W262.13 BOOL  ; B3右伺服位置8设置（HMI）
W262.14 BOOL  ; B3右伺服位置9设置（HMI）
W262.15 BOOL  ; B3右伺服位置10设置（HMI）
W263.00 BOOL  ; B3右伺服待机位手动(HMI)
W263.01 BOOL  ; B3右伺服拨料退回位手动(HMI)
W263.02 BOOL  ; B3右伺服拨料位手动(HMI)
W263.03 BOOL  ; B3右伺服减速位手动(HMI)
W263.04 BOOL  ; B3右伺服等距热压位手动(HMI)
W263.05 BOOL  ; B3右伺服位置6手动(HMI)
W263.06 BOOL  ; B3右伺服位置7手动(HMI)
W263.07 BOOL  ; B3右伺服位置8手动(HMI)
W263.08 BOOL  ; B3右伺服位置9手动(HMI)
W263.09 BOOL  ; B3右伺服位置10手动(HMI)
W263.10 BOOL  ; B3右伺服回原条件
W263.11 BOOL  ; B3右伺服运行锁定
W263.12 BOOL  ; B3右伺服定位条件
W263.13 BOOL  ; B3右伺服回原启动
W263.14 BOOL  ; B3右伺服回原完成
W263.15 BOOL  ; B3右伺服辅助3
W264.00 BOOL  ; B4左伺服回原点手动(HMI)
W264.01 BOOL  ; B4左伺服错误清除(HMI)
W264.02 BOOL  ; B4左伺服JOG高速(HMI)
W264.03 BOOL  ; B4左伺服JOG低速（（HMI）
W264.04 BOOL  ; B4左伺服JOG+（HMI）
W264.05 BOOL  ; B4左伺服JOG-（HMI）
W264.06 BOOL  ; B4左伺服待机位设置（HMI）
W264.07 BOOL  ; B4左伺服拨料退回位设置（HMI）
W264.08 BOOL  ; B4左伺服拨料位设置（HMI）
W264.09 BOOL  ; B4左伺服减速位设置（HMI）
W264.10 BOOL  ; B4左伺服等距热压位设置（HMI）
W264.11 BOOL  ; B4左伺服位置6设置（HMI）
W264.12 BOOL  ; B4左伺服位置7设置（HMI）
W264.13 BOOL  ; B4左伺服位置8设置（HMI）
W264.14 BOOL  ; B4左伺服位置9设置（HMI）
W264.15 BOOL  ; B4左伺服位置10设置（HMI）
W265.00 BOOL  ; B4左伺服待机位手动(HMI)
W265.01 BOOL  ; B4左伺服拨料退回位手动(HMI)
W265.02 BOOL  ; B4左伺服拨料位手动(HMI)
W265.03 BOOL  ; B4左伺服减速位手动(HMI)
W265.04 BOOL  ; B4左伺服等距热压位手动(HMI)
W265.05 BOOL  ; B4左伺服位置6手动(HMI)
W265.06 BOOL  ; B4左伺服位置7手动(HMI)
W265.07 BOOL  ; B4左伺服位置8手动(HMI)
W265.08 BOOL  ; B4左伺服位置9手动(HMI)
W265.09 BOOL  ; B4左伺服位置10手动(HMI)
W265.10 BOOL  ; B4左伺服回原条件
W265.11 BOOL  ; B4左伺服运行锁定
W265.12 BOOL  ; B4左伺服定位条件
W265.13 BOOL  ; B4左伺服回原启动
W265.14 BOOL  ; B4左伺服回原完成
W265.15 BOOL  ; B4左伺服辅助3
W266.00 BOOL  ; B4右伺服回原点手动(HMI)
W266.01 BOOL  ; B4右伺服错误清除(HMI)
W266.02 BOOL  ; B4右伺服JOG高速(HMI)
W266.03 BOOL  ; B4右伺服JOG低速（（HMI）
W266.04 BOOL  ; B4右伺服JOG+（HMI）
W266.05 BOOL  ; B4右伺服JOG-（HMI）
W266.06 BOOL  ; B4右伺服待机位设置（HMI）
W266.07 BOOL  ; B4右伺服拨料退回位设置（HMI）
W266.08 BOOL  ; B4右伺服拨料位设置（HMI）
W266.09 BOOL  ; B4右伺服减速位设置（HMI）
W266.10 BOOL  ; B4右伺服等距热压位设置（HMI）
W266.11 BOOL  ; B4右伺服位置6设置（HMI）
W266.12 BOOL  ; B4右伺服位置7设置（HMI）
W266.13 BOOL  ; B4右伺服位置8设置（HMI）
W266.14 BOOL  ; B4右伺服位置9设置（HMI）
W266.15 BOOL  ; B4右伺服位置10设置（HMI）
W267.00 BOOL  ; B4右伺服待机位手动(HMI)
W267.01 BOOL  ; B4右伺服拨料退回位手动(HMI)
W267.02 BOOL  ; B4右伺服拨料位手动(HMI)
W267.03 BOOL  ; B4右伺服减速位手动(HMI)
W267.04 BOOL  ; B4右伺服等距热压位手动(HMI)
W267.05 BOOL  ; B4右伺服位置6手动(HMI)
W267.06 BOOL  ; B4右伺服位置7手动(HMI)
W267.07 BOOL  ; B4右伺服位置8手动(HMI)
W267.08 BOOL  ; B4右伺服位置9手动(HMI)
W267.09 BOOL  ; B4右伺服位置10手动(HMI)
W267.10 BOOL  ; B4右伺服回原条件
W267.11 BOOL  ; B4右伺服运行锁定
W267.12 BOOL  ; B4右伺服定位条件
W267.13 BOOL  ; B4右伺服回原启动
W267.14 BOOL  ; B4右伺服回原完成
W267.15 BOOL  ; B4右伺服辅助3
W268.00 BOOL  ; 出料伸缩伺服A回原点手动(HMI)
W268.01 BOOL  ; 出料伸缩伺服A错误清除(HMI)
W268.02 BOOL  ; 出料伸缩伺服AJOG高速(HMI)
W268.03 BOOL  ; 出料伸缩伺服AJOG低速（（HMI）
W268.04 BOOL  ; 出料伸缩伺服AJOG+（HMI）
W268.05 BOOL  ; 出料伸缩伺服AJOG-（HMI）
W268.06 BOOL  ; 出料伸缩伺服A位置1设置（HMI）
W268.07 BOOL  ; 出料伸缩伺服A位置2设置（HMI）
W268.08 BOOL  ; 出料伸缩伺服A位置3设置（HMI）
W268.09 BOOL  ; 出料伸缩伺服A位置4设置（HMI）
W268.10 BOOL  ; 出料伸缩伺服A位置5设置（HMI）
W268.11 BOOL  ; 出料伸缩伺服A位置6设置（HMI）
W268.12 BOOL  ; 出料伸缩伺服A位置7设置（HMI）
W268.13 BOOL  ; 出料伸缩伺服A位置8设置（HMI）
W268.14 BOOL  ; 出料伸缩伺服A位置9设置（HMI）
W268.15 BOOL  ; 出料伸缩伺服A位置10设置（HMI）
W269.00 BOOL  ; 出料伸缩伺服A位置1手动(HMI)
W269.01 BOOL  ; 出料伸缩伺服A位置2手动(HMI)
W269.02 BOOL  ; 出料伸缩伺服A位置3手动(HMI)
W269.03 BOOL  ; 出料伸缩伺服A位置4手动(HMI)
W269.04 BOOL  ; 出料伸缩伺服A位置5手动(HMI)
W269.05 BOOL  ; 出料伸缩伺服A位置6手动(HMI)
W269.06 BOOL  ; 出料伸缩伺服A位置7手动(HMI)
W269.07 BOOL  ; 出料伸缩伺服A位置8手动(HMI)
W269.08 BOOL  ; 出料伸缩伺服A位置9手动(HMI)
W269.09 BOOL  ; 出料伸缩伺服A位置10手动(HMI)
W269.10 BOOL  ; 出料伸缩伺服A回原条件
W269.11 BOOL  ; 出料伸缩伺服A运行锁定
W269.12 BOOL  ; 出料伸缩伺服A定位条件
W269.13 BOOL  ; 出料伸缩伺服A回原启动
W269.14 BOOL  ; 出料伸缩伺服A回原完成
W269.15 BOOL  ; 出料伸缩伺服A辅助3
W26.00 BOOL  ; 3ST_进料夹爪上层无料状态正常
W26.01 BOOL  ; 3ST_进料夹爪下层无料状态正常
W26.02 BOOL  ; 3ST_出料夹爪上层无料状态正常
W26.03 BOOL  ; 3ST_出料夹爪下层无料状态正常
W26.04 BOOL  ; 3ST_A出料夹爪A1状态OK
W26.05 BOOL  ; 3ST_A出料夹爪A2状态OK
W26.06 BOOL  ; 3ST_A出料夹爪A3状态OK
W26.07 BOOL  ; 3ST_A出料夹爪A4状态OK
W26.08 BOOL  ; 3ST_A出料夹爪A5状态OK
W26.09 BOOL  ; A1真空正常
W26.10 BOOL  ; A2真空正常
W26.11 BOOL  ; A3真空正常
W26.12 BOOL  ; A4真空正常
W26.13 BOOL  ; A5真空正常
W26.14 BOOL  ; 3ST-A出料夹爪真空正常
W270.00 BOOL  ; 26#伺服回原点手动(HMI)
W270.01 BOOL  ; 26#伺服错误清除(HMI)
W270.02 BOOL  ; 26#伺服JOG高速(HMI)
W270.03 BOOL  ; 26#伺服JOG低速（（HMI）
W270.04 BOOL  ; 26#伺服JOG+（HMI）
W270.05 BOOL  ; 26#伺服JOG-（HMI）
W270.06 BOOL  ; 26#伺服位置1设置（HMI）
W270.07 BOOL  ; 26#伺服位置2设置（HMI）
W270.08 BOOL  ; 26#伺服位置3设置（HMI）
W270.09 BOOL  ; 26#伺服位置4设置（HMI）
W270.10 BOOL  ; 26#伺服位置5设置（HMI）
W270.11 BOOL  ; 26#伺服位置6设置（HMI）
W270.12 BOOL  ; 26#伺服位置7设置（HMI）
W270.13 BOOL  ; 26#伺服位置8设置（HMI）
W270.14 BOOL  ; 26#伺服位置9设置（HMI）
W270.15 BOOL  ; 26#伺服位置10设置（HMI）
W271.00 BOOL  ; 26#伺服位置1手动(HMI)
W271.01 BOOL  ; 26#伺服位置2手动(HMI)
W271.02 BOOL  ; 26#伺服位置3手动(HMI)
W271.03 BOOL  ; 26#伺服位置4手动(HMI)
W271.04 BOOL  ; 26#伺服位置5手动(HMI)
W271.05 BOOL  ; 26#伺服位置6手动(HMI)
W271.06 BOOL  ; 26#伺服位置7手动(HMI)
W271.07 BOOL  ; 26#伺服位置8手动(HMI)
W271.08 BOOL  ; 26#伺服位置9手动(HMI)
W271.09 BOOL  ; 26#伺服位置10手动(HMI)
W271.10 BOOL  ; 26#伺服回原条件
W271.11 BOOL  ; 26#伺服运行锁定
W271.12 BOOL  ; 26#伺服定位条件
W271.13 BOOL  ; 26#伺服回原启动
W271.14 BOOL  ; 26#伺服回原完成
W271.15 BOOL  ; 26#伺服辅助3
W272.00 BOOL  ; 27#左伺服回原点手动(HMI)
W272.01 BOOL  ; 27#左伺服错误清除(HMI)
W272.02 BOOL  ; 27#左伺服JOG高速(HMI)
W272.03 BOOL  ; 27#左伺服JOG低速（（HMI）
W272.04 BOOL  ; 27#左伺服JOG+（HMI）
W272.05 BOOL  ; 27#左伺服JOG-（HMI）
W272.06 BOOL  ; 27#左伺服位置1设置（HMI）
W272.07 BOOL  ; 27#左伺服位置2设置（HMI）
W272.08 BOOL  ; 27#左伺服位置3设置（HMI）
W272.09 BOOL  ; 27#左伺服位置4设置（HMI）
W272.10 BOOL  ; 27#左伺服位置5设置（HMI）
W272.11 BOOL  ; 27#左伺服位置6设置（HMI）
W272.12 BOOL  ; 27#左伺服位置7设置（HMI）
W272.13 BOOL  ; 27#左伺服位置8设置（HMI）
W272.14 BOOL  ; 27#左伺服位置9设置（HMI）
W272.15 BOOL  ; 27#左伺服位置10设置（HMI）
W273.00 BOOL  ; 27#左伺服位置1手动(HMI)
W273.01 BOOL  ; 27#左伺服位置2手动(HMI)
W273.02 BOOL  ; 27#左伺服位置3手动(HMI)
W273.03 BOOL  ; 27#左伺服位置4手动(HMI)
W273.04 BOOL  ; 27#左伺服位置5手动(HMI)
W273.05 BOOL  ; 27#左伺服位置6手动(HMI)
W273.06 BOOL  ; 27#左伺服位置7手动(HMI)
W273.07 BOOL  ; 27#左伺服位置8手动(HMI)
W273.08 BOOL  ; 27#左伺服位置9手动(HMI)
W273.09 BOOL  ; 27#左伺服位置10手动(HMI)
W273.10 BOOL  ; 27#左伺服回原条件
W273.11 BOOL  ; 27#左伺服运行锁定
W273.12 BOOL  ; 27#左伺服定位条件
W273.13 BOOL  ; 27#左伺服回原启动
W273.14 BOOL  ; 27#左伺服回原完成
W273.15 BOOL  ; 27#左伺服辅助3
W274.00 BOOL  ; 接料伺服回原点手动(HMI)
W274.01 BOOL  ; 接料伺服错误清除(HMI)
W274.02 BOOL  ; 接料伺服JOG高速(HMI)
W274.03 BOOL  ; 接料伺服JOG低速（（HMI）
W274.04 BOOL  ; 接料伺服JOG+（HMI）
W274.05 BOOL  ; 接料伺服JOG-（HMI）
W274.06 BOOL  ; 接料伺服出料位设置（HMI）
W274.07 BOOL  ; 接料伺服接料位设置（HMI）
W274.08 BOOL  ; 接料伺服位置3设置（HMI）
W274.09 BOOL  ; 接料伺服位置4设置（HMI）
W274.10 BOOL  ; 接料伺服位置5设置（HMI）
W274.11 BOOL  ; 接料伺服位置6设置（HMI）
W274.12 BOOL  ; 接料伺服位置7设置（HMI）
W274.13 BOOL  ; 接料伺服位置8设置（HMI）
W274.14 BOOL  ; 接料伺服位置9设置（HMI）
W274.15 BOOL  ; 接料伺服位置10设置（HMI）
W275.00 BOOL  ; 接料伺服出料位手动(HMI)
W275.01 BOOL  ; 接料伺服接料位手动(HMI)
W275.02 BOOL  ; 接料伺服位置3手动(HMI)
W275.03 BOOL  ; 接料伺服位置4手动(HMI)
W275.04 BOOL  ; 接料伺服位置5手动(HMI)
W275.05 BOOL  ; 接料伺服位置6手动(HMI)
W275.06 BOOL  ; 接料伺服位置7手动(HMI)
W275.07 BOOL  ; 接料伺服位置8手动(HMI)
W275.08 BOOL  ; 接料伺服位置9手动(HMI)
W275.09 BOOL  ; 接料伺服位置10手动(HMI)
W275.10 BOOL  ; 接料伺服回原条件
W275.11 BOOL  ; 接料伺服运行锁定
W275.12 BOOL  ; 接料伺服定位条件
W275.13 BOOL  ; 接料伺服回原启动
W275.14 BOOL  ; 接料伺服回原完成
W275.15 BOOL  ; 接料伺服辅助3
W27.00 BOOL  ; 3ST_进料夹爪上层有料状态正常
W27.01 BOOL  ; 3ST_进料夹爪下层有料状态正常
W27.02 BOOL  ; 3ST_出料夹爪上层有料状态正常
W27.03 BOOL  ; 3ST_出料夹爪下层有料状态正常
W28.12 BOOL  ; B进料平台允许取料信号
W28.13 BOOL  ; B出料平台允许放料信号
W28.14 BOOL  ; A进料平台允许取料信号
W28.15 BOOL  ; A出料平台允许放料信号
W29.00 BOOL  ; A移栽在上料安全位
W29.01 BOOL  ; 3ST_A移栽在下料安全位
W29.02 BOOL  ; 热压1A有上料需求
W29.03 BOOL  ; 热压2A有上料需求
W29.04 BOOL  ; 热压1A有下料需求
W29.05 BOOL  ; 热压2A有下料需求
W29.06 BOOL  ; 热压1A允许上料
W29.07 BOOL  ; 热压2A允许上料
W29.08 BOOL  ; 热压1A允许下料
W29.09 BOOL  ; 热压2A允许下料
W30.00 BOOL  ; 3ST_B手动切换允许输出标志
W30.01 BOOL  ; 3ST_B自动切换允许输出标志
W30.06 BOOL  ; A边无进料计时
W30.07 BOOL  ; 3ST_A B侧取料
W30.08 BOOL  ; 3ST_B B侧取料
W31.00 BOOL  ; 3ST_B进料夹爪有料标志
W31.01 BOOL  ; 3ST_B进料夹爪无料标志
W31.02 BOOL  ; 3ST_B出料夹爪有料标志
W31.03 BOOL  ; 3ST_B出料夹爪无料标志
W31.09 BOOL  ; B1真空正常
W31.10 BOOL  ; B2真空正常
W31.11 BOOL  ; B3真空正常
W31.12 BOOL  ; B4真空正常
W31.13 BOOL  ; B5真空正常
W31.14 BOOL  ; 3ST-B出料夹爪真空正常
W34.00 BOOL  ; 3ST_B移栽在上料安全位
W34.01 BOOL  ; 3ST_B移栽在下料安全位
W34.02 BOOL  ; 热压1B有上料需求
W34.03 BOOL  ; 热压2B有上料需求
W34.04 BOOL  ; 热压1B有下料需求
W35.00 BOOL  ; 4ST_A手动输出允许
W35.01 BOOL  ; 4ST_A自动输出允许
W35.03 BOOL  ; 4ST_A A侧放料准备(总)
W35.04 BOOL  ; 4ST_A A侧放料允许(总)
W35.05 BOOL  ; 4ST_A A侧取料准备(总)
W35.06 BOOL  ; 4ST_A A侧取料允许(总)
W35.07 BOOL  ; 4ST_A B侧放料准备(总)
W35.08 BOOL  ; 4ST_A B侧放料允许(总)
W35.09 BOOL  ; 4ST_A B侧取料准备(总)
W35.10 BOOL  ; 4ST_A B侧取料允许(总)
W36.00 BOOL  ; 4ST_A所有顶升缩回位
W36.01 BOOL  ; 4ST_A所有顶升伸出位
W36.02 BOOL  ; 4ST_A所有预压退回位
W36.03 BOOL  ; 4ST_A所有预压伸出位
W36.04 BOOL  ; 4ST_A HIP气缸全上位
W36.05 BOOL  ; 4ST_A HIP气缸全下位
W36.06 BOOL  ; 4ST_A气缸全原位
W36.07 BOOL  ; 4ST_A 下压板全A位
W36.08 BOOL  ; 4ST_A 下压板全B位
W36.09 BOOL  ; 4ST_A 侧压伺服均在初始位
W36.10 BOOL  ; 4ST_A 侧压均在拨料退回位
W36.11 BOOL  ; 4ST_A 侧压均在拨料位
W36.12 BOOL  ; 4ST_A 侧压启动&HIP&预压气缸后退条件
W36.13 BOOL  ; 4ST_A 侧压力全部到达区间
W36.14 BOOL  ; 4ST_A HIP全部测试完成
W36.15 BOOL  ; 4ST_A均在拨料等待位
W37.00 BOOL  ; A1 HIP 测试启动
W37.01 BOOL  ; A2 HIP 测试启动
W37.02 BOOL  ; A3 HIP 测试启动
W37.03 BOOL  ; A4 HIP 测试启动
W37.04 BOOL  ; A5 HIP 测试启动
W37.13 BOOL  ; A工位正压压力未超保护值
W37.14 BOOL  ; 替罪羊全在位
W38.00 BOOL  ; 1号A边放料准备1（无其他料）
W38.01 BOOL  ; 1号B边放料准备1（无其他料）
W38.02 BOOL  ; 1号A边放料允许1(无其他料)
W38.03 BOOL  ; 1号B边放料允许1（无其他料）
W38.04 BOOL  ; 4ST_A 1号B边放料准备2（循环）
W38.05 BOOL  ; 4ST_A 1号B边取料准备1（循环）
W38.06 BOOL  ; 4ST_A 1号A边放料准备2（循坏）
W38.07 BOOL  ; 4ST_A 1号A边取料准备1（循环）
W38.08 BOOL  ; 4ST_A 1号B边放料允许2（循环）
W38.09 BOOL  ; 4ST_A 1号B边取料允许1（循环）
W38.10 BOOL  ; 4ST_A 1号A边放料允许2（循坏）
W38.11 BOOL  ; 4ST_A 1号A边取料允许1（循环）
W38.12 BOOL  ; 4ST_A A边取料允许（清料）
W38.13 BOOL  ; 4ST_A B边取料允许（清料）
W38.15 BOOL  ; 顶升安全条件
W39.00 BOOL  ; 4ST-A A边无待热压料
W39.01 BOOL  ; 4ST-A B边无待热压料
W39.02 BOOL  ; 4ST-A 热压无料
W39.03 BOOL  ; 4ST-A B边无完成料
W39.04 BOOL  ; 4ST-A A边无完成料
W39.10 BOOL  ; 4ST-A伺服无异常
W39.14 BOOL  ; 清料条件1
W39.15 BOOL  ; 清料条件2
W400.00 BOOL  ; 前门磁异常
W400.01 BOOL  ; 后门磁异常
W400.02 BOOL  ; 左门磁异常
W400.03 BOOL  ; 右门磁异常
W400.04 BOOL  ; 气源压力开关异常
W400.05 BOOL  ; 主急停按钮异常
W400.06 BOOL  ; 移动屏急停异常
W400.07 BOOL  ; 电脑与PLC连接异常
W400.08 BOOL  ; PLC与副PLC连接异常
W401.00 BOOL  ; 1ST进出料安全光栅异常
W401.01 BOOL  ; 1ST进料定位上层前后松开位异常
W401.02 BOOL  ; 1ST进料定位上层前后夹紧位异常
W401.03 BOOL  ; 1ST进料定位下层前后松开位异常
W401.04 BOOL  ; 1ST进料定位下层前后夹紧位异常
W401.05 BOOL  ; 1ST进料定位上层左右松开位异常
W401.06 BOOL  ; 1ST进料定位上层左右夹紧位异常
W401.07 BOOL  ; 1ST进料定位下层左右松开位异常
W401.08 BOOL  ; 1ST进料定位下层左右夹紧位异常
W401.09 BOOL  ; 1ST进料定位平台上层待料位异常
W401.10 BOOL  ; 1ST进料定位平台上层出料位异常
W401.11 BOOL  ; 1ST进料定位平台下层待料位异常
W401.12 BOOL  ; 1ST进料定位平台下层出料位异常
W401.13 BOOL  ; 1ST进料定位上层有料感应异常
W401.14 BOOL  ; 1ST进料定位下层有料感应异常
W402.00 BOOL  ; 2ST出料定位上层前后松开位异常
W402.01 BOOL  ; 2ST出料定位上层前后夹紧位异常
W402.02 BOOL  ; 2ST出料定位下层前后松开位异常
W402.03 BOOL  ; 2ST出料定位下层前后夹紧位异常
W402.04 BOOL  ; 2ST出料定位上层左右松开位异常
W402.05 BOOL  ; 2ST出料定位上层左右夹紧位异常
W402.06 BOOL  ; 2ST出料定位下层左右松开位异常
W402.07 BOOL  ; 2ST出料定位下层左右夹紧位异常
W402.08 BOOL  ; 2ST出料定位平台上层接料位异常
W402.09 BOOL  ; 2ST出料定位平台上层出料位异常
W402.10 BOOL  ; 2ST出料定位平台下层接料位异常
W402.11 BOOL  ; 2ST出料定位平台下层出料位异常
W402.12 BOOL  ; 2ST出料定位上层有料感应异常
W402.13 BOOL  ; 2ST出料定位下层有料感应异常
W403.00 BOOL  ; 3ST进料夹爪张开位异常
W403.01 BOOL  ; 3ST进料夹爪夹紧位异常
W403.02 BOOL  ; 3ST进料爪上层左压紧上升位异常
W403.03 BOOL  ; 3ST进料爪上层右压紧上升位异常
W403.04 BOOL  ; 3ST进料爪下层左压紧上升位异常
W403.05 BOOL  ; 3ST进料爪下层右压紧上升位异常
W403.06 BOOL  ; 3ST进料爪上层中间压紧上升位异常
W403.07 BOOL  ; 3ST进料爪下层中间压紧上升位异常
W403.08 BOOL  ; 3ST进料夹爪上升位异常
W403.09 BOOL  ; 3ST进料夹爪下降位异常
W403.10 BOOL  ; 3ST进料爪上层有料感应异常
W403.11 BOOL  ; 3ST进料爪下层有料感应异常
W403.12 BOOL  ; 3ST出料夹爪张开位异常
W403.13 BOOL  ; 3ST出料夹爪夹紧位异常
W403.14 BOOL  ; 3ST出料爪上层左压紧上升位异常
W403.15 BOOL  ; 3ST出料爪上层右压紧上升位异常
W404.00 BOOL  ; 3ST出料爪下层左压紧上升位异常
W404.01 BOOL  ; 3ST出料爪下层右压紧上升位异常
W404.02 BOOL  ; 3ST出料夹爪上升位异常
W404.03 BOOL  ; 3ST出料夹爪下降位异常
W404.04 BOOL  ; 3ST出料爪上层有料感应异常
W404.05 BOOL  ; 3ST出料爪下层有料感应异常
W405.00 BOOL  ; 4ST-1热压A增压缸上升位异常
W405.01 BOOL  ; 4ST-1热压A增压缸下降位异常
W405.02 BOOL  ; 4ST-1热压A上层顶升气缸上升位异常
W405.03 BOOL  ; 4ST-1热压A上层顶升气缸下降位异常
W405.04 BOOL  ; 4ST-1热压A下层顶升气缸上升位异常
W405.05 BOOL  ; 4ST-1热压A下层顶升气缸下降位异常
W405.06 BOOL  ; 4ST-1热压A垫高气缸移出位异常
W405.07 BOOL  ; 4ST-1热压A垫高气缸热压位异常
W405.08 BOOL  ; 4ST-1热压A上层Hip测试气缸上升位异常
W405.09 BOOL  ; 4ST-1热压A上层Hip测试气缸下降位异常
W405.10 BOOL  ; 4ST-1热压A下层Hip测试气缸上升位异常
W405.11 BOOL  ; 4ST-1热压A下层Hip测试气缸下降位异常
W405.12 BOOL  ; 4ST-1热压A上层有料感应异常
W405.13 BOOL  ; 4ST-1热压A下层有料感应异常
W405.14 BOOL  ; 4ST-1热压A上层极耳检查异常
W405.15 BOOL  ; 4ST-1热压A下层极耳检查异常
W406.00 BOOL  ; 4ST-1热压A加热跳闸
W407.00 BOOL  ; 4ST-2 热压B增压缸上升位异常
W407.01 BOOL  ; 4ST-2 热压B增压缸下降位异常
W407.02 BOOL  ; 4ST-2 热压B上层顶升气缸上升位异常
W407.03 BOOL  ; 4ST-2 热压B上层顶升气缸下降位异常
W407.04 BOOL  ; 4ST-2 热压B下层顶升气缸上升位异常
W407.05 BOOL  ; 4ST-2 热压B下层顶升气缸下降位异常
W407.06 BOOL  ; 4ST-2 热压B垫高气缸移出位异常
W407.07 BOOL  ; 4ST-2 热压B垫高气缸热压位异常
W407.08 BOOL  ; 4ST-2 热压B上层Hip测试气缸上升位异常
W407.09 BOOL  ; 4ST-2 热压B上层Hip测试气缸下降位异常
W407.10 BOOL  ; 4ST-2 热压B下层Hip测试气缸上升位异常
W407.11 BOOL  ; 4ST-2 热压B下层Hip测试气缸下降位异常
W407.12 BOOL  ; 4ST-2 热压B上层有料感应异常
W407.13 BOOL  ; 4ST-2 热压B下层有料感应异常
W407.14 BOOL  ; 4ST-2 热压B上层极耳检查输入异常
W407.15 BOOL  ; 4ST-2 热压B下层极耳检查输入异常
W408.00 BOOL  ; 4ST-2 热压B加热跳闸
W409.00 BOOL  ; 4ST-3热压C增压缸上升位异常
W409.01 BOOL  ; 4ST-3热压C增压缸下降位异常
W409.02 BOOL  ; 4ST-3热压C上层顶升气缸上升位异常
W409.03 BOOL  ; 4ST-3热压C上层顶升气缸下降位异常
W409.04 BOOL  ; 4ST-3热压C下层顶升气缸上升位异常
W409.05 BOOL  ; 4ST-3热压C下层顶升气缸下降位异常
W409.06 BOOL  ; 4ST-3热压C垫高气缸移出位异常
W409.07 BOOL  ; 4ST-3热压C垫高气缸热压位异常
W409.08 BOOL  ; 4ST-3热压C上层Hip测试气缸上升位异常
W409.09 BOOL  ; 4ST-3热压C上层Hip测试气缸下降位异常
W409.10 BOOL  ; 4ST-3热压C下层Hip测试气缸上升位异常
W409.11 BOOL  ; 4ST-3热压C下层Hip测试气缸下降位异常
W409.12 BOOL  ; 4ST-3热压C上层有料感应异常
W409.13 BOOL  ; 4ST-3热压C下层有料感应异常
W409.14 BOOL  ; 4ST-3热压C上层极耳检查输入异常
W409.15 BOOL  ; 4ST-3热压C下层极耳检查输入异常
W40.00 BOOL  ; 4ST_B手动输出允许
W40.01 BOOL  ; 4ST_B自动输出允许
W40.03 BOOL  ; 4ST_B A侧放料准备(总)
W40.04 BOOL  ; 4ST_B A侧放料允许(总)
W40.04 BOOL  ; 4ST_B A侧放料允许(总)
W40.05 BOOL  ; 4ST_B A侧取料准备(总)
W40.06 BOOL  ; 4ST_B A侧取料允许(总)
W40.06 BOOL  ; 4ST_B A侧取料允许(总)
W40.07 BOOL  ; 4ST_B B侧放料准备(总)
W40.08 BOOL  ; 4ST_B B侧放料允许(总)
W40.08 BOOL  ; 4ST_B B侧放料允许(总)
W40.09 BOOL  ; 4ST_B B侧取料准备(总)
W40.09 BOOL  ; 4ST_B B侧取料准备(总)
W40.10 BOOL  ; 4ST_B B侧取料允许(总)
W40.10 BOOL  ; 4ST_B B侧取料允许(总)
W410.00 BOOL  ; 4ST-3热压C加热跳闸
W411.00 BOOL  ; 3ST进出料转移伺服准备好异常
W411.01 BOOL  ; 3ST进出料转移伺服报警异常
W411.02 BOOL  ; 3ST伸缩伺服准备好异常
W411.03 BOOL  ; 3ST伸缩伺服报警异常
W41.00 BOOL  ; 4ST_B所有顶升缩回位
W41.01 BOOL  ; 4ST_B所有顶升伸出位
W41.02 BOOL  ; 4ST_B所有预压退回位
W41.03 BOOL  ; 4ST_B所有预压伸出位
W41.04 BOOL  ; 4ST_B HIP气缸全上位
W41.05 BOOL  ; 4ST_B HIP气缸全下位
W41.06 BOOL  ; 4ST_B气缸全原位
W41.07 BOOL  ; 4ST_B 下压板全A位
W41.08 BOOL  ; 4ST_B 下压板全B位
W41.09 BOOL  ; 4ST_B 侧压伺服均在初始位
W41.10 BOOL  ; 4ST_B 侧压均在拨料退回位
W41.11 BOOL  ; 4ST_B 侧压均在拨料位
W41.12 BOOL  ; 4ST_B 侧压启动&HIP&预压气缸后退条件
W41.13 BOOL  ; 4ST_B 侧压力全部到达区间
W41.14 BOOL  ; 4ST_B HIP全部测试完成
W41.15 BOOL  ; 4ST_B 侧压均在拨料等待位
W420 CHANNEL  ; 4ST-A报警字1
W421 CHANNEL  ; 4ST-A报警字2
W422 CHANNEL  ; 4ST-A报警字3
W42.00 BOOL  ; B1 HIP 测试启动
W42.01 BOOL  ; B2 HIP 测试启动
W42.02 BOOL  ; B3 HIP 测试启动
W42.03 BOOL  ; B4 HIP 测试启动
W42.04 BOOL  ; B5 HIP 测试启动
W42.13 BOOL  ; B工位正压压力正常
W436.05 BOOL  ; $?St$Bk?_#[481] / 扫码NG满料!!! / $?St$Bk?_#[481]
W436.06 BOOL  ; 扫码NG拉带接近1异常！！！扫码NG拉带位置错误！！！
W436.07 BOOL  ; 扫码NG拉带接近1异常！！！扫码NG拉带位置错误！！！
W437.05 BOOL  ; $?St$Bk?_#[482] / HIPNG满料!!! / $?St$Bk?_#[482]
W437.06 BOOL  ; HIPNG-NG拉带接近1异常！！！HIPNG-NG拉带位置错误！！！
W437.07 BOOL  ; HIPNG-NG拉带接近2异常！！！HIPNG-NG拉带位置错误！！！
W438.05 BOOL  ; $?St$Bk?_#[483] / 工艺NG满料!!! / $?St$Bk?_#[483]
W438.06 BOOL  ; 工艺NG拉带接近1异常！！！工艺NG拉带位置错误！！！
W438.07 BOOL  ; 工艺NG拉带接近2异常！！！工艺NG拉带位置错误！！！
W43.00 BOOL  ; 2号A边放料准备1（无其他料）
W43.01 BOOL  ; 2号B边放料准备1（无其他料）
W43.02 BOOL  ; 2号A边放料允许1(无其他料)
W43.03 BOOL  ; 2号B边放料允许1（无其他料）
W43.04 BOOL  ; 4ST_B 2号B边放料准备2（循环）
W43.05 BOOL  ; 4ST_B 2号B边取料准备1（循环）
W43.06 BOOL  ; 4ST_B 2号A边放料准备2（循坏）
W43.07 BOOL  ; 4ST_B 2号A边取料准备1（循环）
W43.08 BOOL  ; 4ST_B 2号B边放料允许2（循环）
W43.09 BOOL  ; 4ST_B 2号B边取料允许1（循环）
W43.10 BOOL  ; 4ST_B 2号A边放料允许2（循坏）
W43.11 BOOL  ; 4ST_B 2号A边取料允许1（循环）
W43.12 BOOL  ; 4ST_B A边取料允许（清料）
W43.13 BOOL  ; 4ST_B B边取料允许（清料）
W440.00 BOOL  ; $?St$Bk?_#[484] / 7St上层扫码后退感应异常 / $?St$Bk?_#[484]
W440.01 BOOL  ; $?St$Bk?_#[485] / 7St上层扫码前进感应异常 / $?St$Bk?_#[485]
W440.02 BOOL  ; 7St上层扫码缩回感应异常
W440.03 BOOL  ; 7St上层扫码伸出感应异常
W440.04 BOOL  ; 7ST下层扫码后退感应异常
W440.05 BOOL  ; 7ST下层扫码前进感应异常
W440.06 BOOL  ; 7St下层扫码缩回感应异常
W440.07 BOOL  ; 7St下层扫码伸出感应异常
W441.00 BOOL  ; 替罪羊1检测失败
W441.01 BOOL  ; 替罪羊2检测失败
W441.02 BOOL  ; 替罪羊3检测失败
W441.03 BOOL  ; 替罪羊4检测失败
W441.04 BOOL  ; 替罪羊5检测失败
W442.00 BOOL  ; 3ST-A进出料转移A进出料横移伺服A报警异常
W442.01 BOOL  ; 3ST-A进出料转移A进出料伸缩伺服A报警异常
W442.02 BOOL  ; 3ST-A进出料转移A进出料伸缩伺服A1报警异常
W442.03 BOOL  ; 3ST-B进出料转移B进出料横移伺服B报警异常
W442.04 BOOL  ; 3ST-B进出料转移B进出料伸缩伺服B报警异常
W442.05 BOOL  ; 3ST-B进出料转移B进出料伸缩伺服B1报警异常
W442.06 BOOL  ; 4ST-A热压A正压伺服A报警异常
W442.07 BOOL  ; 4ST-A热压A压板平移伺服A报警异常
W442.08 BOOL  ; 4ST-A热压A侧压A1左伺服报警异常
W442.09 BOOL  ; 4ST-A热压A侧压A1右伺服报警异常
W442.10 BOOL  ; 4ST-A热压A侧压A2左伺服报警异常
W442.11 BOOL  ; 4ST-A热压A侧压A2右伺服报警异常
W442.12 BOOL  ; 4ST-A热压A侧压A3左伺服报警异常
W442.13 BOOL  ; 4ST-A热压A侧压A3右伺服报警异常
W442.14 BOOL  ; 4ST-A热压A侧压A4左伺服报警异常
W442.15 BOOL  ; 4ST-A热压A侧压A4右伺服报警异常
W443.00 BOOL  ; 4ST-A热压A侧压A5左伺服报警异常
W443.01 BOOL  ; 4ST-A热压A侧压A5右伺服报警异常
W443.02 BOOL  ; 4ST-B热压B正压伺服B报警异常
W443.03 BOOL  ; 4ST-B热压B压板平移伺服B报警异常
W443.04 BOOL  ; 4ST-B热压B侧压B1左伺服报警异常
W443.05 BOOL  ; 4ST-B热压B侧压B1右伺服报警异常
W443.06 BOOL  ; 4ST-B热压B侧压B2左伺服报警异常
W443.07 BOOL  ; 4ST-B热压B侧压B2右伺服报警异常
W443.08 BOOL  ; 4ST-B热压B侧压B3左伺服报警异常
W443.09 BOOL  ; 4ST-B热压B侧压B3右伺服报警异常
W443.10 BOOL  ; 4ST-B热压B侧压B4左伺服报警异常
W443.11 BOOL  ; 4ST-B热压B侧压B4右伺服报警异常
W443.12 BOOL  ; 4ST-B热压B侧压B5左伺服报警异常
W443.13 BOOL  ; 4ST-B热压B侧压B5右伺服报警异常
W443.14 BOOL  ; 7ST接料扫码接料伺服READY异常
W443.15 BOOL  ; 7ST接料扫码接料伺服报警异常
W444.00 BOOL  ; 进出料横移伺服A回原点未完成
W444.01 BOOL  ; 进出料伸缩伺服A回原点未完成
W444.02 BOOL  ; 进出料横移伺服B回原点未完成
W444.03 BOOL  ; 进出料伸缩伺服B回原点未完成
W444.04 BOOL  ; 正压伺服A回原点未完成
W444.05 BOOL  ; 压板平移伺服A回原点未完成
W444.06 BOOL  ; 侧压A1左伺服回原未完成
W444.07 BOOL  ; 侧压A1右伺服回原点未完成
W444.08 BOOL  ; 侧压A2左伺服回原点未完成
W444.09 BOOL  ; 侧压A2右伺服回原点未完成
W444.10 BOOL  ; 侧压A3左伺服回原点未完成
W444.11 BOOL  ; 侧压A3右伺服回原点未完成
W444.12 BOOL  ; 侧压A4左伺服回原点未完成
W444.13 BOOL  ; 侧压A4右伺服回原点未完成
W444.14 BOOL  ; 正压伺服B回原点未完成
W444.15 BOOL  ; 压板平移伺服B回原点未完成
W445.00 BOOL  ; 侧压B1左伺服回原点未完成
W445.01 BOOL  ; 侧压B1右伺服回原点未完成
W445.02 BOOL  ; 侧压B2左伺服回原点未完成
W445.03 BOOL  ; 侧压B2右伺服回原点未完成
W445.04 BOOL  ; 侧压B3左伺服回原点未完成
W445.05 BOOL  ; 侧压B3右伺服回原点未完成
W445.06 BOOL  ; 侧压B4左伺服回原点未完成
W445.07 BOOL  ; 侧压B4右伺服回原点未完成
W445.11 BOOL  ; 接料伺服回原点未完成
W446.00 BOOL  ; 进出料伸缩伺服A未在初始位
W446.01 BOOL  ; 上料定位A未在垂直位
W446.02 BOOL  ; A进出料夹爪机构未在上升位
W446.03 BOOL  ; 下料定位A未在垂直位
W446.04 BOOL  ; A进料夹爪机构不在上位
W446.05 BOOL  ; A进料夹爪不在下位
W446.07 BOOL  ; A进料夹爪不在上位
W446.08 BOOL  ; A出料夹爪机构不在上位
W446.09 BOOL  ; A出料夹爪不在上位
W446.10 BOOL  ; A出料夹爪不在下位
W447.00 BOOL  ; 进出料伸缩伺服B未在初始位
W447.01 BOOL  ; 上料定位B未在垂直位
W447.02 BOOL  ; B进出料夹爪机构未在上升位
W447.03 BOOL  ; 下料定位B未在垂直位
W447.04 BOOL  ; B进料夹爪机构不在上位
W447.05 BOOL  ; B进料夹爪不在下位
W447.07 BOOL  ; B进料夹爪不在上位
W447.08 BOOL  ; B出料夹爪机构不在上位
W447.09 BOOL  ; B出料夹爪不在上位
W447.10 BOOL  ; B出料夹爪不在下位
W448.00 BOOL  ; 4ST-A正压A1压力超保护
W448.01 BOOL  ; 4ST-A正压A2压力超保护
W448.02 BOOL  ; 4ST-A正压A3压力超保护
W448.03 BOOL  ; 4ST-A正压A4压力超保护
W448.04 BOOL  ; 4ST-A正压A5压力超保护
W448.05 BOOL  ; 4ST-A侧压A1左超保护
W448.06 BOOL  ; 4ST-A侧压A1右超保护
W448.07 BOOL  ; 4ST-A侧压A2左超保护
W448.08 BOOL  ; 4ST-A侧压A2右超保护
W448.09 BOOL  ; 4ST-A侧压A3左超保护
W448.10 BOOL  ; 4ST-A侧压A3右超保护
W448.11 BOOL  ; 4ST-A侧压A4左超保护
W448.12 BOOL  ; 4ST-A侧压A4右超保护
W448.13 BOOL  ; 4ST-A侧压A5左超保护
W448.14 BOOL  ; 4ST-A侧压A5右超保护
W449.00 BOOL  ; 4ST-B正压B1压力超保护
W449.01 BOOL  ; 4ST-B正压B2压力超保护
W449.02 BOOL  ; 4ST-B正压B3压力超保护
W449.03 BOOL  ; 4ST-B正压B4压力超保护
W449.04 BOOL  ; 4ST-B正压B5压力超保护
W449.05 BOOL  ; 4ST-B侧压B1左超保护
W449.06 BOOL  ; 4ST-B侧压B1右超保护
W449.07 BOOL  ; 4ST-B侧压B2左超保护
W449.08 BOOL  ; 4ST-B侧压B2右超保护
W449.09 BOOL  ; 4ST-B侧压B3左超保护
W449.10 BOOL  ; 4ST-B侧压B3右超保护
W449.11 BOOL  ; 4ST-B侧压B4左超保护
W449.12 BOOL  ; 4ST-B侧压B4右超保护
W449.13 BOOL  ; 4ST-B侧压B5左超保护
W449.14 BOOL  ; 4ST-B侧压B5右超保护
W44.00 BOOL  ; 4ST-B A边无待热压料
W44.01 BOOL  ; 4ST-B B边无待热压料
W44.02 BOOL  ; 4ST-B 热压无料
W44.03 BOOL  ; 4ST-B B边无完成料
W44.04 BOOL  ; 4ST-B A边无完成料
W44.14 BOOL  ; 清料条件1
W44.15 BOOL  ; 清料条件2
W451.00 BOOL  ; 前门磁1异常
W451.01 BOOL  ; 前门磁2异常
W451.02 BOOL  ; 前门磁3异常
W451.03 BOOL  ; 前门磁4异常
W451.04 BOOL  ; 前门磁5异常
W451.05 BOOL  ; 前门磁6异常
W451.06 BOOL  ; 前门磁7异常
W451.07 BOOL  ; 后门磁1异常
W451.08 BOOL  ; 后门磁2异常
W451.09 BOOL  ; 后门磁3异常
W451.10 BOOL  ; 后门磁4异常
W451.11 BOOL  ; 后门磁5异常
W451.12 BOOL  ; 后门磁6异常
W451.13 BOOL  ; 后门磁7异常
W451.14 BOOL  ; 前侧急停异常
W451.15 BOOL  ; 后侧急停异常
W45.00 BOOL  ; 5ST-A手动允许输出
W45.01 BOOL  ; 5ST-A自动允许输出
W480 CHANNEL  ; 热压A1测试结果(解析位)
W481 CHANNEL  ; 热压A1测试结果
W482 CHANNEL  ; 热压A2测试结果
W483 CHANNEL  ; 热压A2测试结果
W484 CHANNEL  ; 热压A3测试结果
W485 CHANNEL  ; 热压A3测试结果
W486 CHANNEL  ; 热压A4测试结果
W487 CHANNEL  ; 热压A4测试结果
W488 CHANNEL  ; 热压A1测试结果
W490 CHANNEL  ; 热压B1测试结果
W491 CHANNEL  ; 热压B1测试结果
W492 CHANNEL  ; 热压B2测试结果
W493 CHANNEL  ; 热压B2测试结果
W494 CHANNEL  ; 热压B3测试结果
W495 CHANNEL  ; 热压B3测试结果
W496 CHANNEL  ; 热压B4测试结果
W497 CHANNEL  ; 热压B4测试结果
W498 CHANNEL  ; 热压A测试结果_9
W50.00 BOOL  ; 5ST-B手动允许输出
W50.01 BOOL  ; 5ST-B自动允许输出
W55.00 BOOL  ; 6ST手动切换允许输出标志
W55.01 BOOL  ; 6ST自动切换允许输出标志
W55.02 BOOL  ; 机器人初始化(HMI)
W55.03 BOOL  ; 应抓A平台
W55.04 BOOL  ; 应抓B平台
W55.05 BOOL  ; 机器人初始化1:停止程序
W55.06 BOOL  ; 机器人初始化2:清除报警
W55.07 BOOL  ; 机器人初始化3:程序复位
W55.08 BOOL  ; 机器人初始化4:程序启动
W55.09 BOOL  ; $?St$Bk?_#[486] / 取A平台条件 / $?St$Bk?_#[486]
W55.10 BOOL  ; $?St$Bk?_#[487] / 取B平台条件 / $?St$Bk?_#[487]
W55.11 BOOL  ; $?St$Bk?_#[488] / 下料机器人柔性报警 / $?St$Bk?_#[488]
W55.12 BOOL  ; $?St$Bk?_#[489] / 机器人初始化(复位) / $?St$Bk?_#[489]
W55.13 BOOL  ; $?St$Bk?_#[490] / 模拟可放料信号-下游 / $?St$Bk?_#[490]
W55.14 BOOL  ; $?St$Bk?_#[491] / 工艺NG拉带启动辅助 / $?St$Bk?_#[491]
W55.15 BOOL  ; $?St$Bk?_#[492] / HipotNG拉带启动辅助 / $?St$Bk?_#[492]
W56 CHANNEL  ; 下料机器人任务信息
W56.00 BOOL  ; 下料任务辅助1
W56.01 BOOL  ; 下料任务辅助2
W56.02 BOOL  ; 下料任务辅助3
W56.03 BOOL  ; 下料任务辅助4
W56.04 BOOL  ; 下料任务辅助5
W57 CHANNEL  ; 下料机器人位置信息
W57.00 BOOL  ; 下料R位置辅助1
W57.01 BOOL  ; 下料R位置辅助2
W57.02 BOOL  ; 下料R位置辅助3
W57.03 BOOL  ; 下料R位置辅助4
W58.00 BOOL  ; 抓料上位A(01)
W58.01 BOOL  ; 抓料位A(02)
W58.02 BOOL  ; 抓料上位B(03)
W58.03 BOOL  ; 抓料位B(04)
W58.04 BOOL  ; 放料上位(05)
W58.05 BOOL  ; 放料位(06)
W58.06 BOOL  ; 工艺NG上位1(20)
W58.07 BOOL  ; 工艺NG位1(21)
W58.08 BOOL  ; HipotNG上位1(30)
W58.09 BOOL  ; HipotNG位1(31)
W58.10 BOOL  ; 任意上位
W59 CHANNEL  ; 下料机器人夹爪状态正确
W59.00 BOOL  ; R夹爪1状态正确
W59.01 BOOL  ; R夹爪2状态正确
W59.02 BOOL  ; R夹爪3状态正确
W59.03 BOOL  ; R夹爪4状态正确
W59.04 BOOL  ; R夹爪5状态正确
W60.00 BOOL  ; 7ST手动切换允许输出标志
W60.01 BOOL  ; 7ST自动切换允许输出标志
W60.02 BOOL  ; $?St$Bk?_#[493] / 模拟设备放料完成-上游 / $?St$Bk?_#[493]
W60.03 BOOL  ; 强制可放料信号-上游
W60.04 BOOL  ; 模拟设备在安全位-上游
W60.05 BOOL  ; 模拟设备放料完成-上游
W60.06 BOOL  ; 手动上层扫码
W60.07 BOOL  ; 手动上层扫码(M)
W60.08 BOOL  ; 自动上层扫码(A)
W60.09 BOOL  ; 上层扫码输出
W60.10 BOOL  ; 手动下层扫码
W60.11 BOOL  ; 手动下层扫码(M)
W60.12 BOOL  ; 自动下层扫码(A)
W60.13 BOOL  ; 下层扫码输出
W61.00 BOOL  ; 扫码数据传输成功1
W61.01 BOOL  ; 扫码数据传输成功2
W61.02 BOOL  ; 扫码数据传输成功3
W61.03 BOOL  ; 扫码数据传输成功4
W61.04 BOOL  ; 扫码数据传输成功5
W61.05 BOOL  ; 扫码数据传输成功6
W61.06 BOOL  ; 扫码数据传输成功7
W61.07 BOOL  ; 扫码数据传输成功8
W61.08 BOOL  ; 扫码数据传输成功9
W61.09 BOOL  ; 扫码数据传输成功10
W65.01 BOOL  ; 1St记忆清除按钮(HMI)
W65.02 BOOL  ; 2StA进料定位平台记忆清除(HMI)
W65.03 BOOL  ; 2StB进料定位平台记忆清除(HMI)
W65.04 BOOL  ; 3A记忆清除（T）
W65.05 BOOL  ; 3B记忆清除（T）
W65.06 BOOL  ; 4A记忆清除（T）
W65.07 BOOL  ; 4B记忆清除（T）
W65.08 BOOL  ; 5StA出料定位平台记忆清除(HMI)
W65.09 BOOL  ; 5StB出料定位平台记忆清除(HMI)
W65.10 BOOL  ; 6St下料机器人记忆清除按钮(HMI)
W65.11 BOOL  ; 7St接料机构记忆清除(HMI)
W80 CHANNEL  ; 1#副PLC读写步骤
W81 CHANNEL  ; 2#副PLC读写步骤
W82 CHANNEL  ; 3#副PLC读写步骤
W8.00 BOOL  ; 端口都没忙
W8.01 BOOL  ; 写入条件
W8.02 BOOL  ; ST5520_通讯全测试状态
W8.03 BOOL  ; 全测试条件
W8.04 BOOL  ; ST5520_参数全写入状态
W8.05 BOOL  ; 断开全测试
W8.06 BOOL  ; 断开全写入
W8.10 BOOL  ; 复位
W8.12 BOOL  ; 手动测试
W98 CHANNEL  ; 伺服错误清除字
W98.00 BOOL  ; 轴1错误清除
W98.01 BOOL  ; 轴2错误清除
H_AF1_R H_Pit_Read_Resistance_Value
H_AF2_R H_Pit_Read_Resistance_Value
NC433_0 _NCx600_Setting
NC433_0_2000_X_Home _NCx051A_Home_DINT
NC433_0_2000_X_Pos01 _NCx011A_MoveAbsolute_DINT
NC433_0_2000_X_Pos02 _NCx011A_MoveAbsolute_DINT
NC433_0_2000_X_Pos03 _NCx011A_MoveAbsolute_DINT
NC433_0_2000_X_Pos04 _NCx011A_MoveAbsolute_DINT
NC433_0_2000_X_Pos05 _NCx011A_MoveAbsolute_DINT
NC433_0_2000_X_Pos06 _NCx011A_MoveAbsolute_DINT
NC433_0_2000_X_Pos07 _NCx011A_MoveAbsolute_DINT
NC433_0_2000_X_Pos08 _NCx011A_MoveAbsolute_DINT
NC433_0_2000_Y_Home _NCx051A_Home_DINT
NC433_0_2000_Y_Pos01 _NCx011A_MoveAbsolute_DINT
NC433_0_2000_Y_Pos02 _NCx011A_MoveAbsolute_DINT
NC433_0_2000_Y_Pos03 _NCx011A_MoveAbsolute_DINT
P_2141 P_change
P_2142 P_change
P_2143 P_change
P_2144 P_change
P_2145 P_change
P_2146 P_change

## Program MAIN (cyclic task 0)
Local symbols
D6020D6316 UDINT

### Section 系统运行

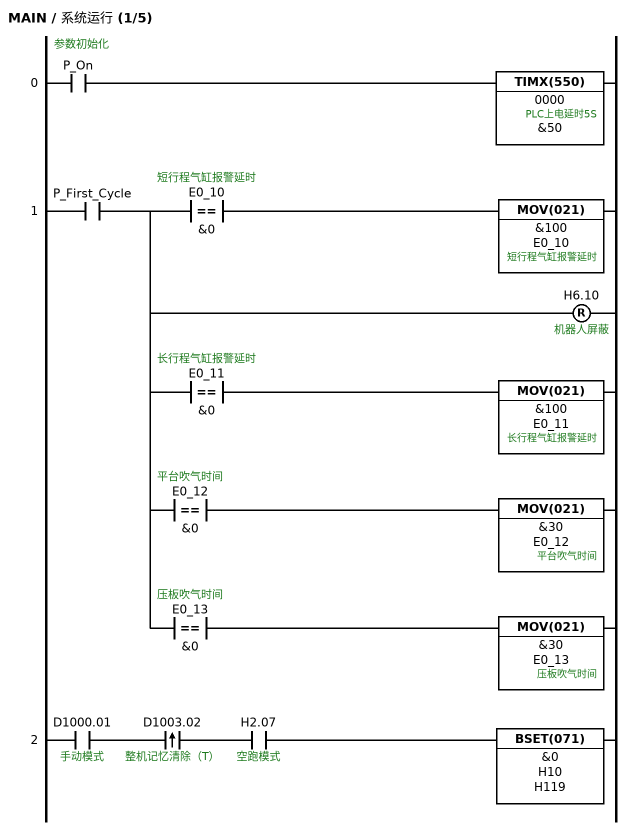
; rung 0: 参数初始化
LD P_On
TIMX(550) 0000 &50  ; PLC上电延时5S
; rung 1
LD P_First_Cycle
OUT TR0
AND=(300) E0_10 &0  ; 短行程气缸报警延时
MOV(021) &100 E0_10  ; 短行程气缸报警延时
LD TR0
RSET H6.10  ; 机器人屏蔽
AND=(300) E0_11 &0  ; 长行程气缸报警延时
MOV(021) &100 E0_11  ; 长行程气缸报警延时
LD TR0
AND=(300) E0_12 &0  ; 平台吹气时间
MOV(021) &30 E0_12  ; 平台吹气时间
LD TR0
AND=(300) E0_13 &0  ; 压板吹气时间
MOV(021) &30 E0_13  ; 压板吹气时间
; rung 2
LD D1000.01  ; 手动模式
@AND D1003.02  ; 整机记忆清除（T）
AND H2.07  ; 空跑模式
BSET(071) &0 H10 H119

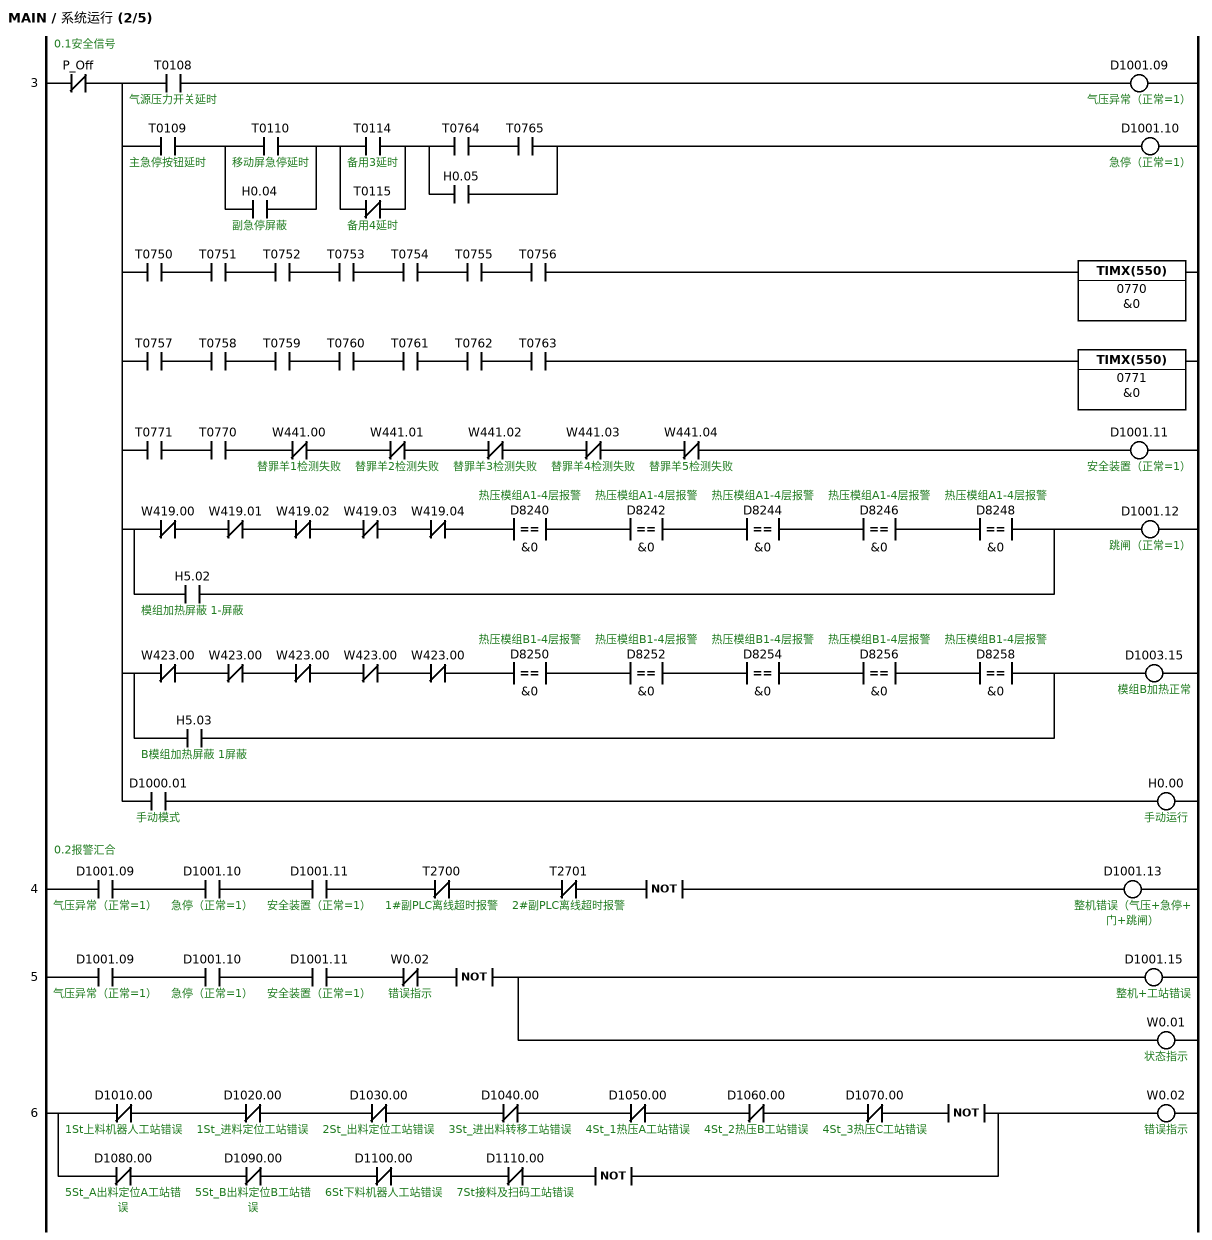
; rung 3: 0.1安全信号
LDNOT P_Off
OUT TR0
AND T0108  ; 气源压力开关延时
OUT D1001.09  ; 气压异常（正常=1）
LD TR0
AND T0109  ; 主急停按钮延时
LD T0110  ; 移动屏急停延时
OR H0.04  ; 副急停屏蔽
ANDLD
LD T0114  ; 备用3延时
ORNOT T0115  ; 备用4延时
ANDLD
LD T0764
AND T0765
OR H0.05
ANDLD
OUT D1001.10  ; 急停（正常=1）
LD TR0
AND T0750
AND T0751
AND T0752
AND T0753
AND T0754
AND T0755
AND T0756
TIMX(550) 0770 &0
LD TR0
AND T0757
AND T0758
AND T0759
AND T0760
AND T0761
AND T0762
AND T0763
TIMX(550) 0771 &0
LD TR0
AND T0771
AND T0770
ANDNOT W441.00  ; 替罪羊1检测失败
ANDNOT W441.01  ; 替罪羊2检测失败
ANDNOT W441.02  ; 替罪羊3检测失败
ANDNOT W441.03  ; 替罪羊4检测失败
ANDNOT W441.04  ; 替罪羊5检测失败
OUT D1001.11  ; 安全装置（正常=1）
LD TR0
LDNOT W419.00
ANDNOT W419.01
ANDNOT W419.02
ANDNOT W419.03
ANDNOT W419.04
AND=L(301) D8240 &0  ; 热压模组A1-4层报警
AND=L(301) D8242 &0  ; 热压模组A1-4层报警
AND=L(301) D8244 &0  ; 热压模组A1-4层报警
AND=L(301) D8246 &0  ; 热压模组A1-4层报警
AND=L(301) D8248 &0  ; 热压模组A1-4层报警
OR H5.02  ; 模组加热屏蔽 1-屏蔽
ANDLD
OUT D1001.12  ; 跳闸（正常=1）
LD TR0
LDNOT W423.00
ANDNOT W423.00
ANDNOT W423.00
ANDNOT W423.00
ANDNOT W423.00
AND=L(301) D8250 &0  ; 热压模组B1-4层报警
AND=L(301) D8252 &0  ; 热压模组B1-4层报警
AND=L(301) D8254 &0  ; 热压模组B1-4层报警
AND=L(301) D8256 &0  ; 热压模组B1-4层报警
AND=L(301) D8258 &0  ; 热压模组B1-4层报警
OR H5.03  ; B模组加热屏蔽 1屏蔽
ANDLD
OUT D1003.15  ; 模组B加热正常
LD TR0
AND D1000.01  ; 手动模式
OUT H0.00  ; 手动运行
; rung 4: 0.2报警汇合
LD D1001.09  ; 气压异常（正常=1）
AND D1001.10  ; 急停（正常=1）
AND D1001.11  ; 安全装置（正常=1）
ANDNOT T2700  ; 1#副PLC离线超时报警
ANDNOT T2701  ; 2#副PLC离线超时报警
NOT(520)
OUT D1001.13  ; 整机错误（气压+急停+门+跳闸）
; rung 5
LD D1001.09  ; 气压异常（正常=1）
AND D1001.10  ; 急停（正常=1）
AND D1001.11  ; 安全装置（正常=1）
ANDNOT W0.02  ; 错误指示
NOT(520)
OUT D1001.15  ; 整机+工站错误
OUT W0.01  ; 状态指示
; rung 6
LDNOT D1010.00  ; 1St上料机器人工站错误
ANDNOT D1020.00  ; 1St_进料定位工站错误
ANDNOT D1030.00  ; 2St_出料定位工站错误
ANDNOT D1040.00  ; 3St_进出料转移工站错误
ANDNOT D1050.00  ; 4St_1热压A工站错误
ANDNOT D1060.00  ; 4St_2热压B工站错误
ANDNOT D1070.00  ; 4St_3热压C工站错误
NOT(520)
LDNOT D1080.00  ; 5St_A出料定位A工站错误
ANDNOT D1090.00  ; 5St_B出料定位B工站错误
ANDNOT D1100.00  ; 6St下料机器人工站错误
ANDNOT D1110.00  ; 7St接料及扫码工站错误
NOT(520)
ORLD
OUT W0.02  ; 错误指示

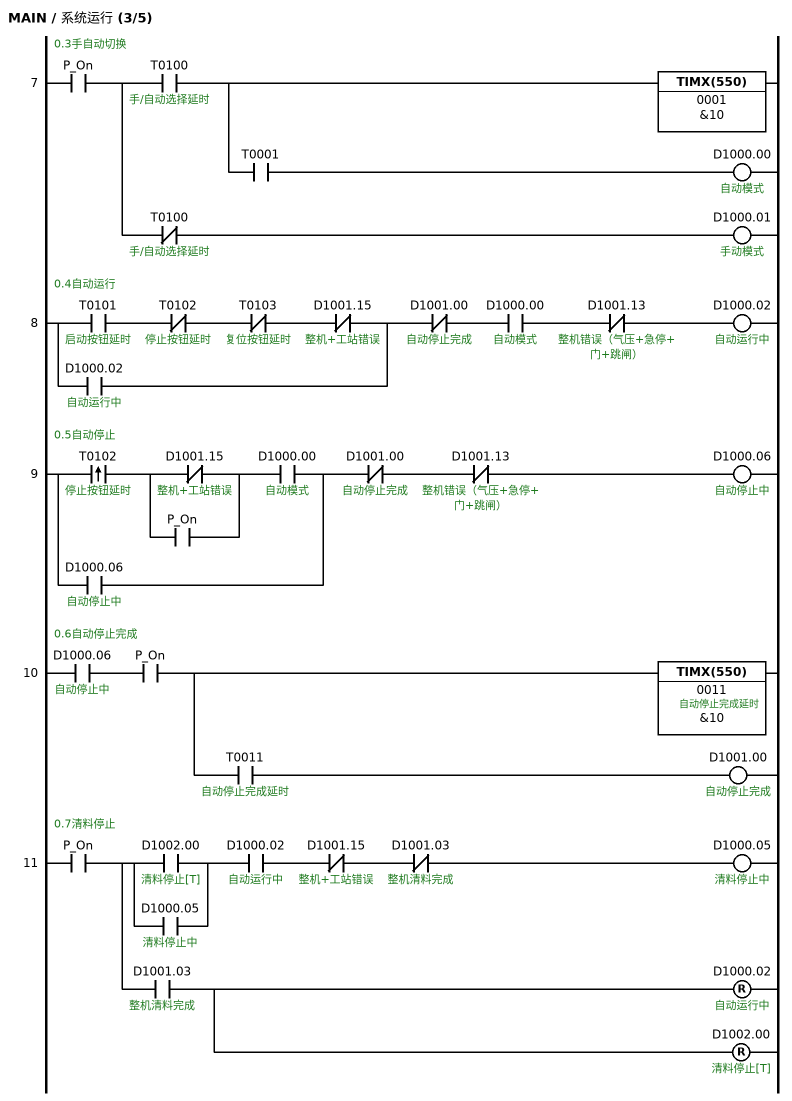
; rung 7: 0.3手自动切换
LD P_On
OUT TR0
AND T0100  ; 手/自动选择延时
TIMX(550) 0001 &10
AND T0001
OUT D1000.00  ; 自动模式
LD TR0
ANDNOT T0100  ; 手/自动选择延时
OUT D1000.01  ; 手动模式
; rung 8: 0.4自动运行
LD T0101  ; 启动按钮延时
ANDNOT T0102  ; 停止按钮延时
ANDNOT T0103  ; 复位按钮延时
ANDNOT D1001.15  ; 整机+工站错误
OR D1000.02  ; 自动运行中
ANDNOT D1001.00  ; 自动停止完成
AND D1000.00  ; 自动模式
ANDNOT D1001.13  ; 整机错误（气压+急停+门+跳闸）
OUT D1000.02  ; 自动运行中
; rung 9: 0.5自动停止
@LD T0102  ; 停止按钮延时
LDNOT D1001.15  ; 整机+工站错误
OR P_On
ANDLD
AND D1000.00  ; 自动模式
OR D1000.06  ; 自动停止中
ANDNOT D1001.00  ; 自动停止完成
ANDNOT D1001.13  ; 整机错误（气压+急停+门+跳闸）
OUT D1000.06  ; 自动停止中
; rung 10: 0.6自动停止完成
LD D1000.06  ; 自动停止中
AND P_On
TIMX(550) 0011 &10  ; 自动停止完成延时
AND T0011  ; 自动停止完成延时
OUT D1001.00  ; 自动停止完成
; rung 11: 0.7清料停止
LD P_On
OUT TR0
LD D1002.00  ; 清料停止[T]
OR D1000.05  ; 清料停止中
ANDLD
AND D1000.02  ; 自动运行中
ANDNOT D1001.15  ; 整机+工站错误
ANDNOT D1001.03  ; 整机清料完成
OUT D1000.05  ; 清料停止中
LD TR0
AND D1001.03  ; 整机清料完成
RSET D1000.02  ; 自动运行中
RSET D1002.00  ; 清料停止[T]

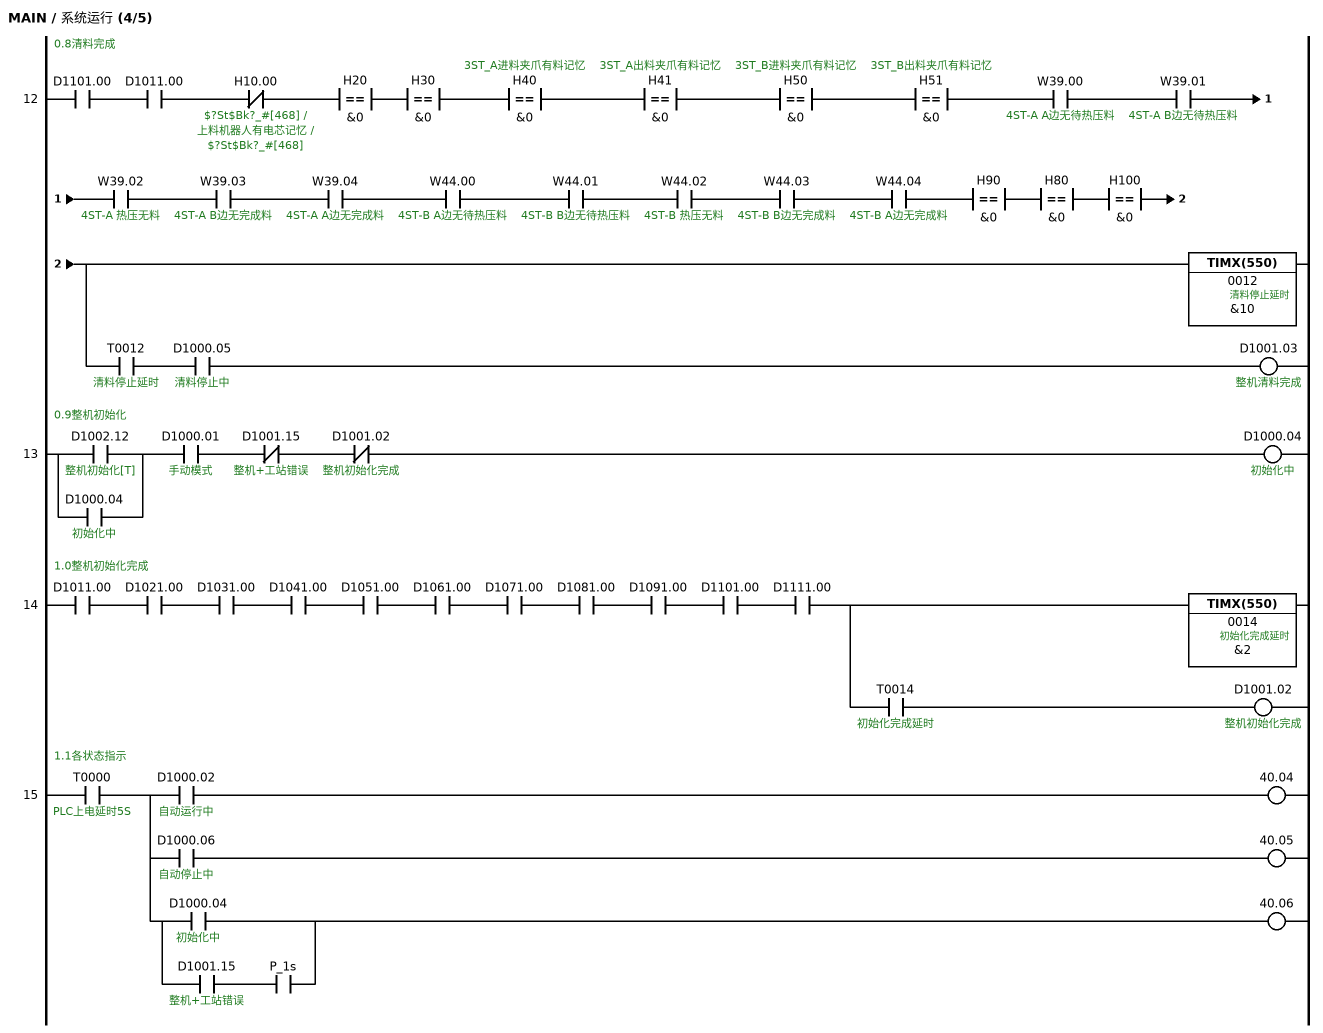
; rung 12: 0.8清料完成
LD D1101.00
AND D1011.00
ANDNOT H10.00  ; $?St$Bk?_#[468] / 上料机器人有电芯记忆 / $?St$Bk?_#[468]
AND=(300) H20 &0
AND=(300) H30 &0
AND=(300) H40 &0  ; 3ST_A进料夹爪有料记忆
AND=(300) H41 &0  ; 3ST_A出料夹爪有料记忆
AND=(300) H50 &0  ; 3ST_B进料夹爪有料记忆
AND=(300) H51 &0  ; 3ST_B出料夹爪有料记忆
AND W39.00  ; 4ST-A A边无待热压料
AND W39.01  ; 4ST-A B边无待热压料
AND W39.02  ; 4ST-A 热压无料
AND W39.03  ; 4ST-A B边无完成料
AND W39.04  ; 4ST-A A边无完成料
AND W44.00  ; 4ST-B A边无待热压料
AND W44.01  ; 4ST-B B边无待热压料
AND W44.02  ; 4ST-B 热压无料
AND W44.03  ; 4ST-B B边无完成料
AND W44.04  ; 4ST-B A边无完成料
AND=(300) H90 &0
AND=(300) H80 &0
AND=(300) H100 &0
TIMX(550) 0012 &10  ; 清料停止延时
AND T0012  ; 清料停止延时
AND D1000.05  ; 清料停止中
OUT D1001.03  ; 整机清料完成
; rung 13: 0.9整机初始化
LD D1002.12  ; 整机初始化[T]
OR D1000.04  ; 初始化中
AND D1000.01  ; 手动模式
ANDNOT D1001.15  ; 整机+工站错误
ANDNOT D1001.02  ; 整机初始化完成
OUT D1000.04  ; 初始化中
; rung 14: 1.0整机初始化完成
LD D1011.00
AND D1021.00
AND D1031.00
AND D1041.00
AND D1051.00
AND D1061.00
AND D1071.00
AND D1081.00
AND D1091.00
AND D1101.00
AND D1111.00
TIMX(550) 0014 &2  ; 初始化完成延时
AND T0014  ; 初始化完成延时
OUT D1001.02  ; 整机初始化完成
; rung 15: 1.1各状态指示
LD T0000  ; PLC上电延时5S
OUT TR0
AND D1000.02  ; 自动运行中
OUT 40.04
LD TR0
AND D1000.06  ; 自动停止中
OUT 40.05
LD TR0
LD D1000.04  ; 初始化中
LD D1001.15  ; 整机+工站错误
AND P_1s
ORLD
ANDLD
OUT 40.06

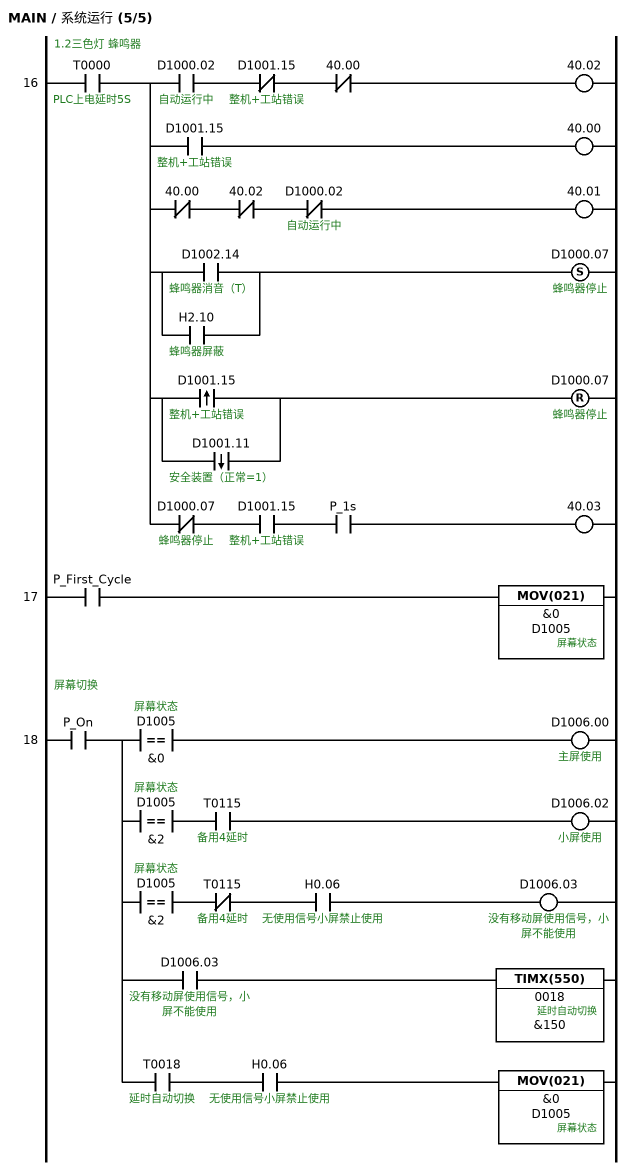
; rung 16: 1.2三色灯 蜂鸣器
LD T0000  ; PLC上电延时5S
OUT TR0
AND D1000.02  ; 自动运行中
ANDNOT D1001.15  ; 整机+工站错误
ANDNOT 40.00
OUT 40.02
LD TR0
AND D1001.15  ; 整机+工站错误
OUT 40.00
LD TR0
ANDNOT 40.00
ANDNOT 40.02
ANDNOT D1000.02  ; 自动运行中
OUT 40.01
LD TR0
LD D1002.14  ; 蜂鸣器消音（T）
OR H2.10  ; 蜂鸣器屏蔽
ANDLD
SET D1000.07  ; 蜂鸣器停止
LD TR0
@LD D1001.15  ; 整机+工站错误
%OR D1001.11  ; 安全装置（正常=1）
ANDLD
RSET D1000.07  ; 蜂鸣器停止
LD TR0
ANDNOT D1000.07  ; 蜂鸣器停止
AND D1001.15  ; 整机+工站错误
AND P_1s
OUT 40.03
; rung 17
LD P_First_Cycle
MOV(021) &0 D1005  ; 屏幕状态
; rung 18: 屏幕切换
LD P_On
OUT TR0
AND=(300) D1005 &0  ; 屏幕状态
OUT D1006.00  ; 主屏使用
LD TR0
AND=(300) D1005 &2  ; 屏幕状态
AND T0115  ; 备用4延时
OUT D1006.02  ; 小屏使用
LD TR0
AND=(300) D1005 &2  ; 屏幕状态
ANDNOT T0115  ; 备用4延时
AND H0.06  ; 无使用信号小屏禁止使用
OUT D1006.03  ; 没有移动屏使用信号，小屏不能使用
LD TR0
AND D1006.03  ; 没有移动屏使用信号，小屏不能使用
TIMX(550) 0018 &150  ; 延时自动切换
LD TR0
AND T0018  ; 延时自动切换
AND H0.06  ; 无使用信号小屏禁止使用
MOV(021) &0 D1005  ; 屏幕状态

### Section NC433_0_2000

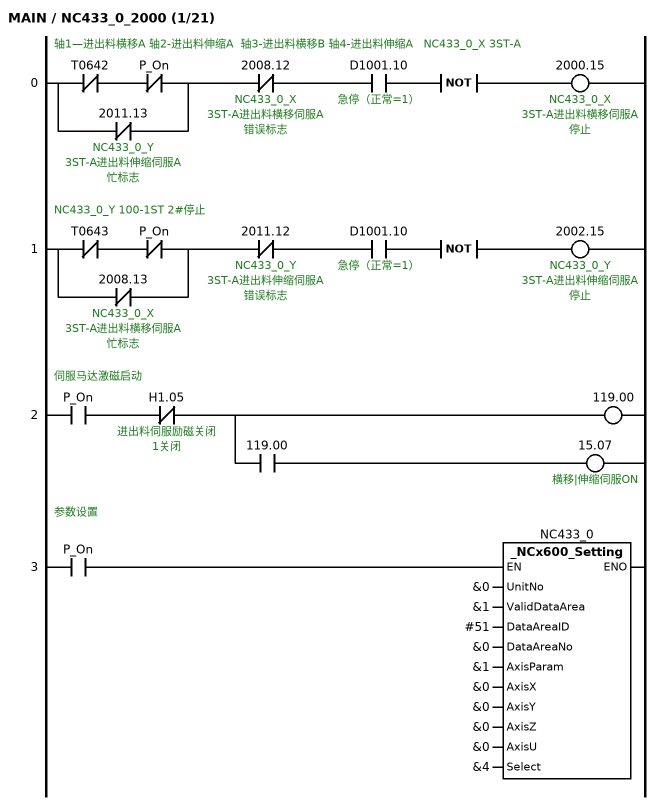
; rung 0: 轴1—进出料横移A 轴2-进出料伸缩A  轴3-进出料横移B 轴4-进出料伸缩A   NC433_0_X 3ST-A
LDNOT T0642
ANDNOT P_On
ORNOT 2011.13  ; NC433_0_Y 3ST-A进出料伸缩伺服A忙标志
ANDNOT 2008.12  ; NC433_0_X 3ST-A进出料横移伺服A错误标志
AND D1001.10  ; 急停（正常=1）
NOT(520)
OUT 2000.15  ; NC433_0_X 3ST-A进出料横移伺服A停止
; rung 1: NC433_0_Y 100-1ST 2#停止
LDNOT T0643
ANDNOT P_On
ORNOT 2008.13  ; NC433_0_X 3ST-A进出料横移伺服A忙标志
ANDNOT 2011.12  ; NC433_0_Y 3ST-A进出料伸缩伺服A错误标志
AND D1001.10  ; 急停（正常=1）
NOT(520)
OUT 2002.15  ; NC433_0_Y 3ST-A进出料伸缩伺服A停止
; rung 2: 伺服马达激磁启动
LD P_On
ANDNOT H1.05  ; 进出料伺服励磁关闭 1关闭
OUT 119.00
AND 119.00
OUT 15.07  ; 横移|伸缩伺服ON
; rung 3: 参数设置
LD P_On
CALL NC433_0 : _NCx600_Setting (UnitNo := &0, ValidDataArea := &1, DataAreaID := #51, DataAreaNo := &0, AxisParam := &1, AxisX := &0, AxisY := &0, AxisZ := &0, AxisU := &0, Select := &4)

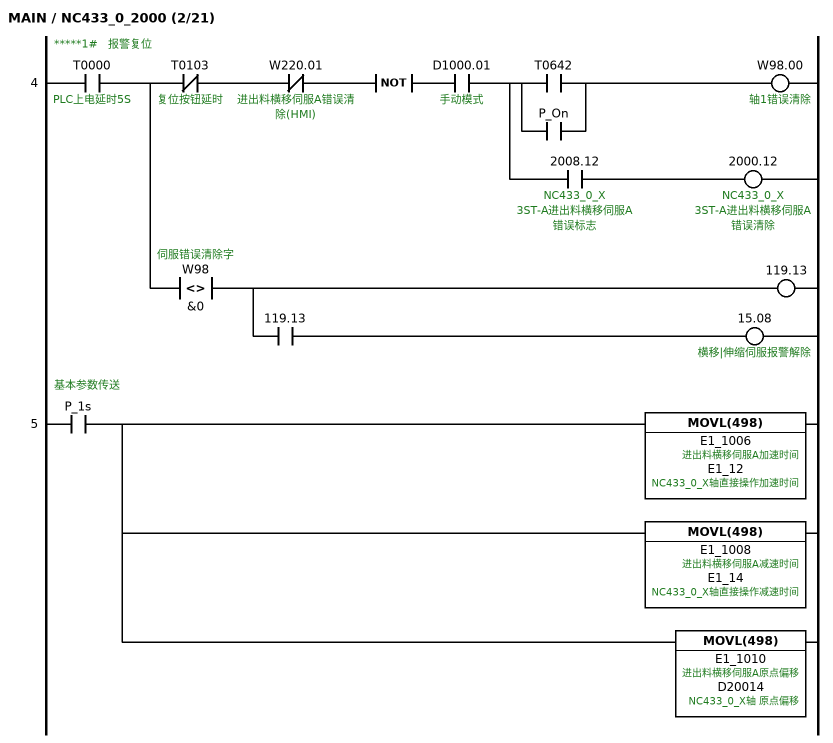
; rung 4: *****1#   报警复位
LD T0000  ; PLC上电延时5S
OUT TR0
ANDNOT T0103  ; 复位按钮延时
ANDNOT W220.01  ; 进出料横移伺服A错误清除(HMI)
NOT(520)
AND D1000.01  ; 手动模式
OUT TR1
LD T0642
OR P_On
ANDLD
OUT W98.00  ; 轴1错误清除
LD TR1
AND 2008.12  ; NC433_0_X 3ST-A进出料横移伺服A错误标志
OUT 2000.12  ; NC433_0_X 3ST-A进出料横移伺服A错误清除
LD TR0
AND<>L(306) W98 &0  ; 伺服错误清除字
OUT 119.13
AND 119.13
OUT 15.08  ; 横移|伸缩伺服报警解除
; rung 5: 基本参数传送
LD P_1s
MOVL(498) E1_1006 E1_12  ; 进出料横移伺服A加速时间, NC433_0_X轴直接操作加速时间
MOVL(498) E1_1008 E1_14  ; 进出料横移伺服A减速时间, NC433_0_X轴直接操作减速时间
MOVL(498) E1_1010 D20014  ; 进出料横移伺服A原点偏移, NC433_0_X轴 原点偏移

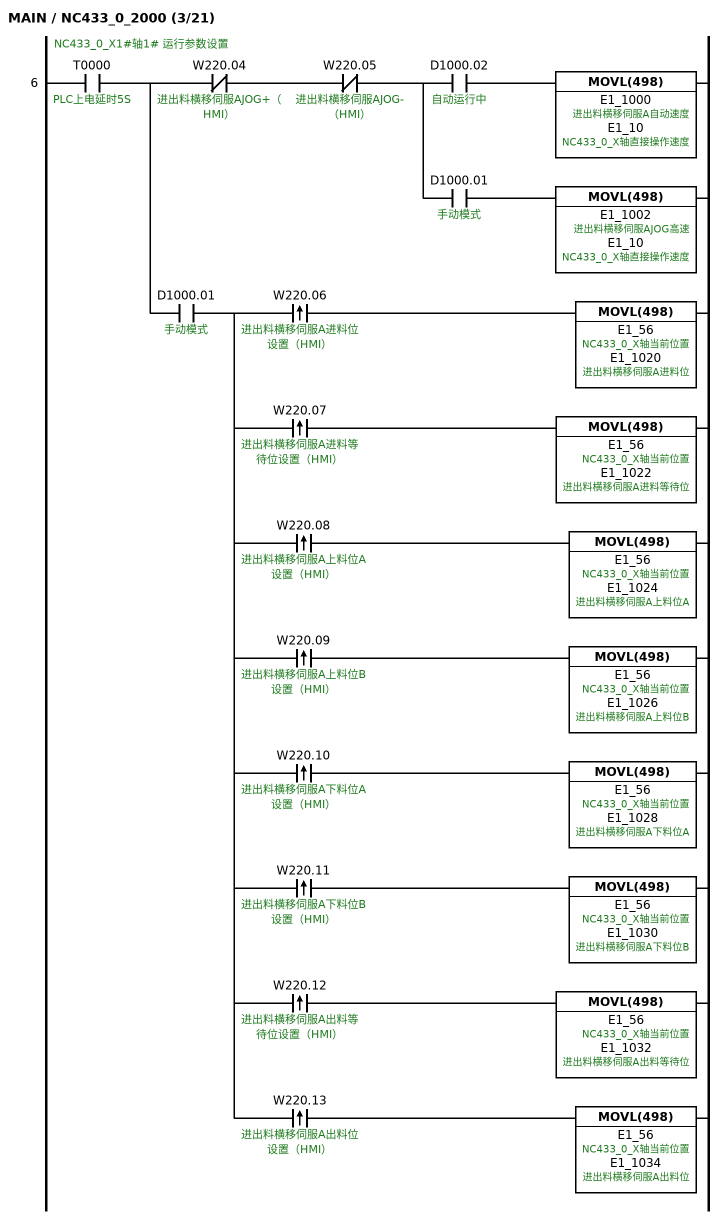
; rung 6: NC433_0_X1#轴1# 运行参数设置
LD T0000  ; PLC上电延时5S
OUT TR0
ANDNOT W220.04  ; 进出料横移伺服AJOG+（HMI）
ANDNOT W220.05  ; 进出料横移伺服AJOG-（HMI）
OUT TR1
AND D1000.02  ; 自动运行中
MOVL(498) E1_1000 E1_10  ; 进出料横移伺服A自动速度, NC433_0_X轴直接操作速度
LD TR1
AND D1000.01  ; 手动模式
MOVL(498) E1_1002 E1_10  ; 进出料横移伺服AJOG高速, NC433_0_X轴直接操作速度
LD TR0
AND D1000.01  ; 手动模式
OUT TR0
@AND W220.06  ; 进出料横移伺服A进料位设置（HMI）
MOVL(498) E1_56 E1_1020  ; NC433_0_X轴当前位置, 进出料横移伺服A进料位
LD TR0
@AND W220.07  ; 进出料横移伺服A进料等待位设置（HMI）
MOVL(498) E1_56 E1_1022  ; NC433_0_X轴当前位置, 进出料横移伺服A进料等待位
LD TR0
@AND W220.08  ; 进出料横移伺服A上料位A设置（HMI）
MOVL(498) E1_56 E1_1024  ; NC433_0_X轴当前位置, 进出料横移伺服A上料位A
LD TR0
@AND W220.09  ; 进出料横移伺服A上料位B设置（HMI）
MOVL(498) E1_56 E1_1026  ; NC433_0_X轴当前位置, 进出料横移伺服A上料位B
LD TR0
@AND W220.10  ; 进出料横移伺服A下料位A设置（HMI）
MOVL(498) E1_56 E1_1028  ; NC433_0_X轴当前位置, 进出料横移伺服A下料位A
LD TR0
@AND W220.11  ; 进出料横移伺服A下料位B设置（HMI）
MOVL(498) E1_56 E1_1030  ; NC433_0_X轴当前位置, 进出料横移伺服A下料位B
LD TR0
@AND W220.12  ; 进出料横移伺服A出料等待位设置（HMI）
MOVL(498) E1_56 E1_1032  ; NC433_0_X轴当前位置, 进出料横移伺服A出料等待位
LD TR0
@AND W220.13  ; 进出料横移伺服A出料位设置（HMI）
MOVL(498) E1_56 E1_1034  ; NC433_0_X轴当前位置, 进出料横移伺服A出料位

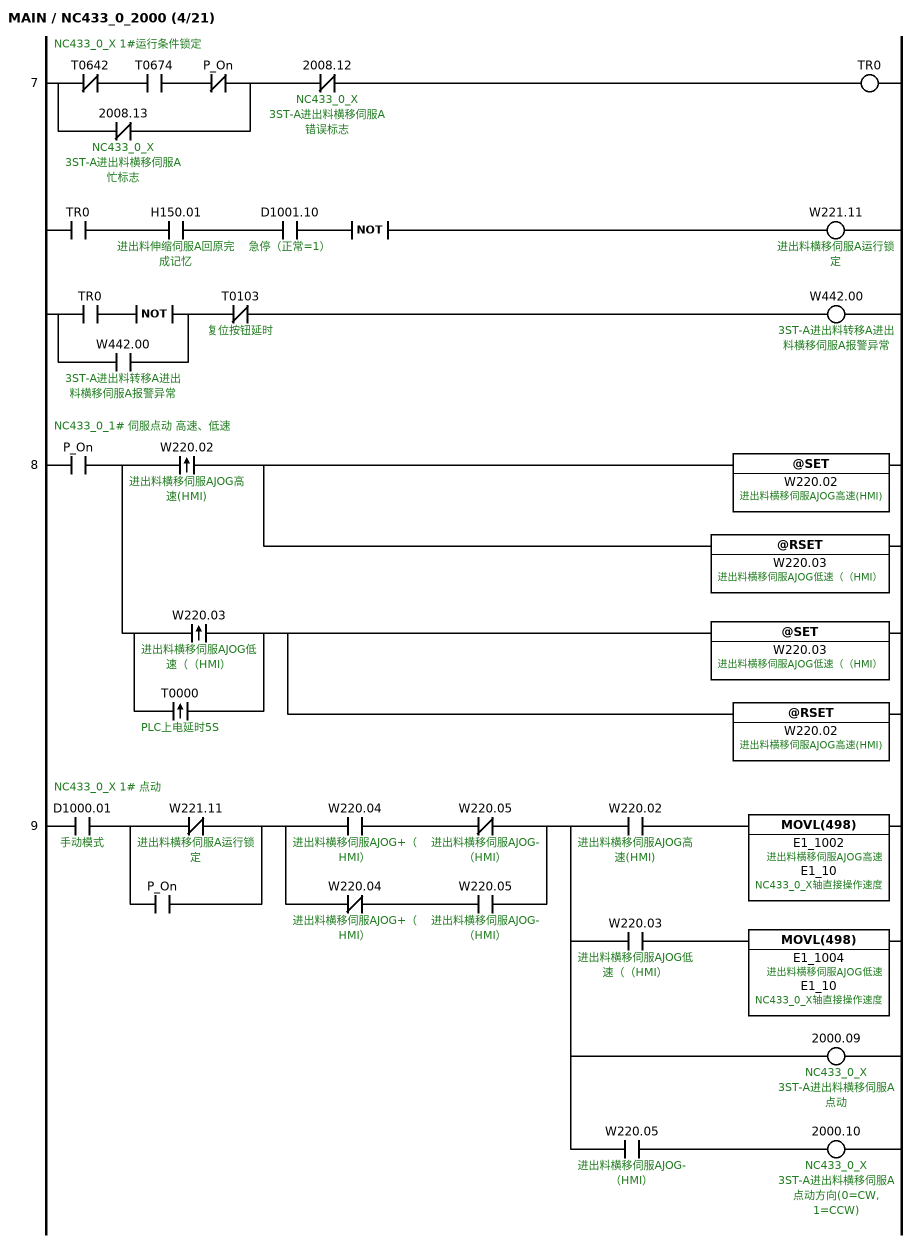
; rung 7: NC433_0_X 1#运行条件锁定
LDNOT T0642
AND T0674
ANDNOT P_On
ORNOT 2008.13  ; NC433_0_X 3ST-A进出料横移伺服A忙标志
ANDNOT 2008.12  ; NC433_0_X 3ST-A进出料横移伺服A错误标志
OUT TR0
AND H150.01  ; 进出料伸缩伺服A回原完成记忆
AND D1001.10  ; 急停（正常=1）
NOT(520)
OUT W221.11  ; 进出料横移伺服A运行锁定
LD TR0
NOT(520)
OR W442.00  ; 3ST-A进出料转移A进出料横移伺服A报警异常
ANDNOT T0103  ; 复位按钮延时
OUT W442.00  ; 3ST-A进出料转移A进出料横移伺服A报警异常
; rung 8: NC433_0_1# 伺服点动 高速、低速
LD P_On
OUT TR0
@AND W220.02  ; 进出料横移伺服AJOG高速(HMI)
@SET W220.02  ; 进出料横移伺服AJOG高速(HMI)
@RSET W220.03  ; 进出料横移伺服AJOG低速（（HMI）
LD TR0
@LD W220.03  ; 进出料横移伺服AJOG低速（（HMI）
@OR T0000  ; PLC上电延时5S
ANDLD
@SET W220.03  ; 进出料横移伺服AJOG低速（（HMI）
@RSET W220.02  ; 进出料横移伺服AJOG高速(HMI)
; rung 9: NC433_0_X 1# 点动
LD D1000.01  ; 手动模式
LDNOT W221.11  ; 进出料横移伺服A运行锁定
OR P_On
ANDLD
LD W220.04  ; 进出料横移伺服AJOG+（HMI）
ANDNOT W220.05  ; 进出料横移伺服AJOG-（HMI）
LDNOT W220.04  ; 进出料横移伺服AJOG+（HMI）
AND W220.05  ; 进出料横移伺服AJOG-（HMI）
ORLD
ANDLD
OUT TR0
AND W220.02  ; 进出料横移伺服AJOG高速(HMI)
MOVL(498) E1_1002 E1_10  ; 进出料横移伺服AJOG高速, NC433_0_X轴直接操作速度
LD TR0
AND W220.03  ; 进出料横移伺服AJOG低速（（HMI）
MOVL(498) E1_1004 E1_10  ; 进出料横移伺服AJOG低速, NC433_0_X轴直接操作速度
LD TR0
OUT 2000.09  ; NC433_0_X 3ST-A进出料横移伺服A点动
AND W220.05  ; 进出料横移伺服AJOG-（HMI）
OUT 2000.10  ; NC433_0_X 3ST-A进出料横移伺服A点动方向(0=CW,1=CCW)

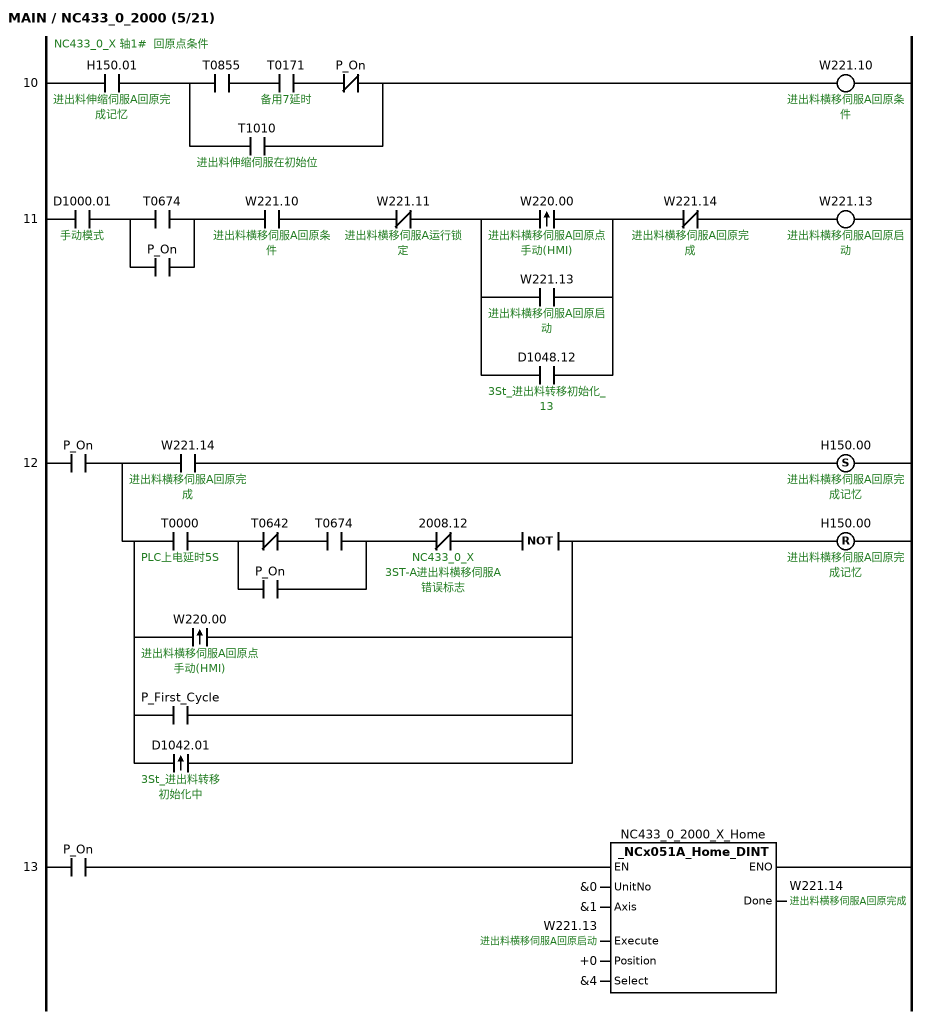
; rung 10: NC433_0_X 轴1#  回原点条件
LD H150.01  ; 进出料伸缩伺服A回原完成记忆
LD T0855
AND T0171  ; 备用7延时
ANDNOT P_On
OR T1010  ; 进出料伸缩伺服在初始位
ANDLD
OUT W221.10  ; 进出料横移伺服A回原条件
; rung 11
LD D1000.01  ; 手动模式
LD T0674
OR P_On
ANDLD
AND W221.10  ; 进出料横移伺服A回原条件
ANDNOT W221.11  ; 进出料横移伺服A运行锁定
@LD W220.00  ; 进出料横移伺服A回原点手动(HMI)
OR W221.13  ; 进出料横移伺服A回原启动
OR D1048.12  ; 3St_进出料转移初始化_13
ANDLD
ANDNOT W221.14  ; 进出料横移伺服A回原完成
OUT W221.13  ; 进出料横移伺服A回原启动
; rung 12
LD P_On
OUT TR0
AND W221.14  ; 进出料横移伺服A回原完成
SET H150.00  ; 进出料横移伺服A回原完成记忆
LD TR0
LD T0000  ; PLC上电延时5S
LDNOT T0642
AND T0674
OR P_On
ANDLD
ANDNOT 2008.12  ; NC433_0_X 3ST-A进出料横移伺服A错误标志
NOT(520)
@OR W220.00  ; 进出料横移伺服A回原点手动(HMI)
OR P_First_Cycle
@OR D1042.01  ; 3St_进出料转移 初始化中
ANDLD
RSET H150.00  ; 进出料横移伺服A回原完成记忆
; rung 13
LD P_On
CALL NC433_0_2000_X_Home : _NCx051A_Home_DINT (UnitNo := &0, Axis := &1, Execute := W221.13, Position := +0, Select := &4, Done => W221.14)  ; 进出料横移伺服A回原启动, 进出料横移伺服A回原完成

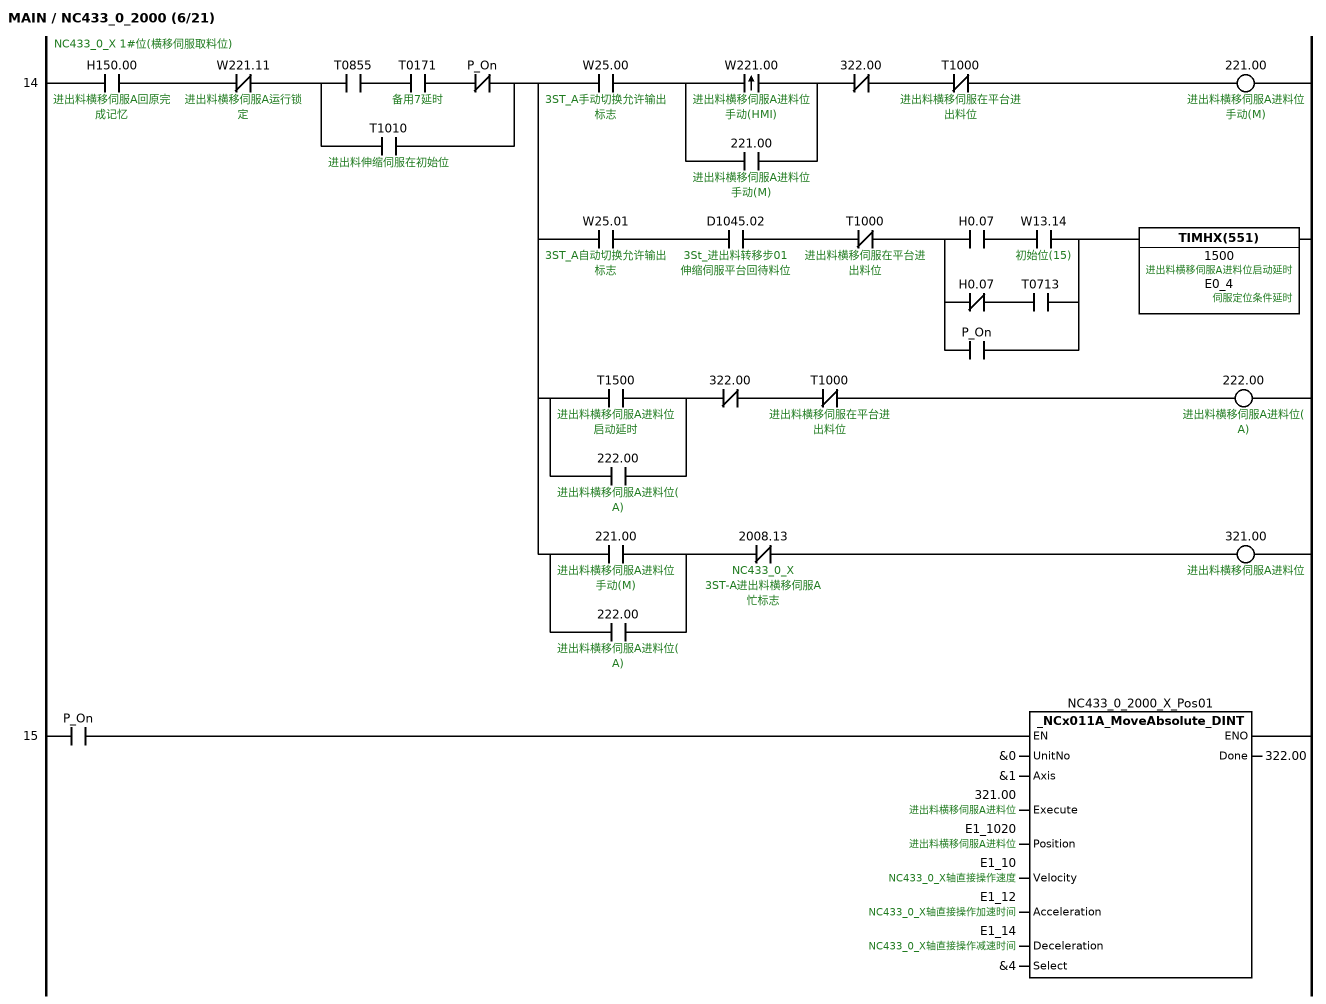
; rung 14: NC433_0_X 1#位(横移伺服取料位)
LD H150.00  ; 进出料横移伺服A回原完成记忆
ANDNOT W221.11  ; 进出料横移伺服A运行锁定
LD T0855
AND T0171  ; 备用7延时
ANDNOT P_On
OR T1010  ; 进出料伸缩伺服在初始位
ANDLD
OUT TR0
AND W25.00  ; 3ST_A手动切换允许输出标志
@LD W221.00  ; 进出料横移伺服A进料位手动(HMI)
OR 221.00  ; 进出料横移伺服A进料位手动(M)
ANDLD
ANDNOT 322.00
ANDNOT T1000  ; 进出料横移伺服在平台进出料位
OUT 221.00  ; 进出料横移伺服A进料位手动(M)
LD TR0
AND W25.01  ; 3ST_A自动切换允许输出标志
AND D1045.02  ; 3St_进出料转移步01 伸缩伺服平台回待料位
ANDNOT T1000  ; 进出料横移伺服在平台进出料位
LD H0.07
AND W13.14  ; 初始位(15)
LDNOT H0.07
AND T0713
ORLD
OR P_On
ANDLD
TIMHX(551) 1500 E0_4  ; 伺服定位条件延时, 进出料横移伺服A进料位启动延时
LD TR0
LD T1500  ; 进出料横移伺服A进料位启动延时
OR 222.00  ; 进出料横移伺服A进料位(A)
ANDLD
ANDNOT 322.00
ANDNOT T1000  ; 进出料横移伺服在平台进出料位
OUT 222.00  ; 进出料横移伺服A进料位(A)
LD TR0
LD 221.00  ; 进出料横移伺服A进料位手动(M)
OR 222.00  ; 进出料横移伺服A进料位(A)
ANDLD
ANDNOT 2008.13  ; NC433_0_X 3ST-A进出料横移伺服A忙标志
OUT 321.00  ; 进出料横移伺服A进料位
; rung 15
LD P_On
CALL NC433_0_2000_X_Pos01 : _NCx011A_MoveAbsolute_DINT (UnitNo := &0, Axis := &1, Execute := 321.00, Position := E1_1020, Velocity := E1_10, Acceleration := E1_12, Deceleration := E1_14, Select := &4, Done => 322.00)  ; 进出料横移伺服A进料位, NC433_0_X轴直接操作速度, NC433_0_X轴直接操作加速时间, NC433_0_X轴直接操作减速时间

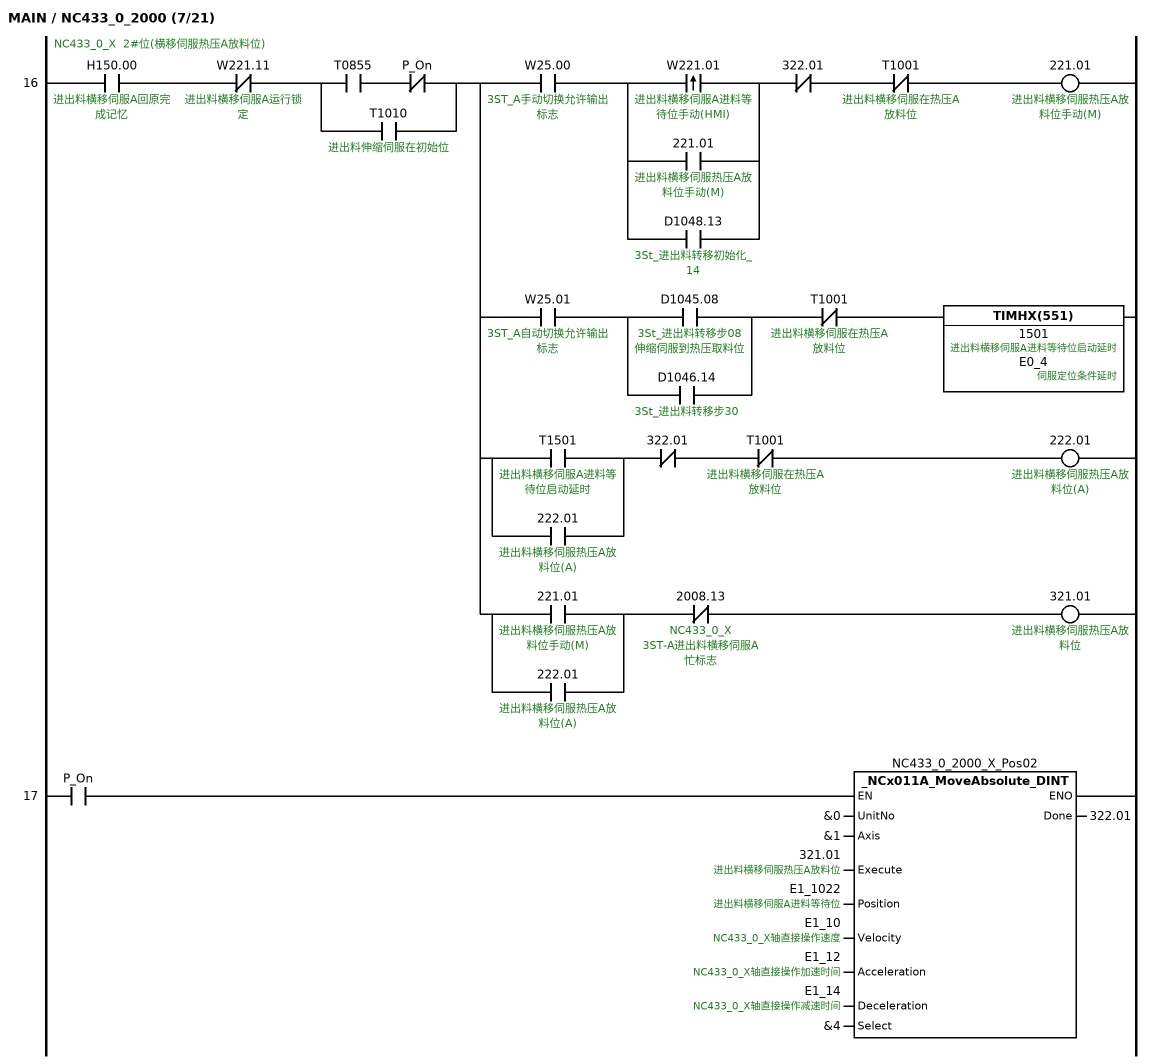
; rung 16: NC433_0_X  2#位(横移伺服热压A放料位)
LD H150.00  ; 进出料横移伺服A回原完成记忆
ANDNOT W221.11  ; 进出料横移伺服A运行锁定
LD T0855
ANDNOT P_On
OR T1010  ; 进出料伸缩伺服在初始位
ANDLD
OUT TR0
AND W25.00  ; 3ST_A手动切换允许输出标志
@LD W221.01  ; 进出料横移伺服A进料等待位手动(HMI)
OR 221.01  ; 进出料横移伺服热压A放料位手动(M)
OR D1048.13  ; 3St_进出料转移初始化_14
ANDLD
ANDNOT 322.01
ANDNOT T1001  ; 进出料横移伺服在热压A放料位
OUT 221.01  ; 进出料横移伺服热压A放料位手动(M)
LD TR0
AND W25.01  ; 3ST_A自动切换允许输出标志
LD D1045.08  ; 3St_进出料转移步08 伸缩伺服到热压取料位
OR D1046.14  ; 3St_进出料转移步30
ANDLD
ANDNOT T1001  ; 进出料横移伺服在热压A放料位
TIMHX(551) 1501 E0_4  ; 伺服定位条件延时, 进出料横移伺服A进料等待位启动延时
LD TR0
LD T1501  ; 进出料横移伺服A进料等待位启动延时
OR 222.01  ; 进出料横移伺服热压A放料位(A)
ANDLD
ANDNOT 322.01
ANDNOT T1001  ; 进出料横移伺服在热压A放料位
OUT 222.01  ; 进出料横移伺服热压A放料位(A)
LD TR0
LD 221.01  ; 进出料横移伺服热压A放料位手动(M)
OR 222.01  ; 进出料横移伺服热压A放料位(A)
ANDLD
ANDNOT 2008.13  ; NC433_0_X 3ST-A进出料横移伺服A忙标志
OUT 321.01  ; 进出料横移伺服热压A放料位
; rung 17
LD P_On
CALL NC433_0_2000_X_Pos02 : _NCx011A_MoveAbsolute_DINT (UnitNo := &0, Axis := &1, Execute := 321.01, Position := E1_1022, Velocity := E1_10, Acceleration := E1_12, Deceleration := E1_14, Select := &4, Done => 322.01)  ; 进出料横移伺服热压A放料位, 进出料横移伺服A进料等待位, NC433_0_X轴直接操作速度, NC433_0_X轴直接操作加速时间, NC433_0_X轴直接操作减速时间

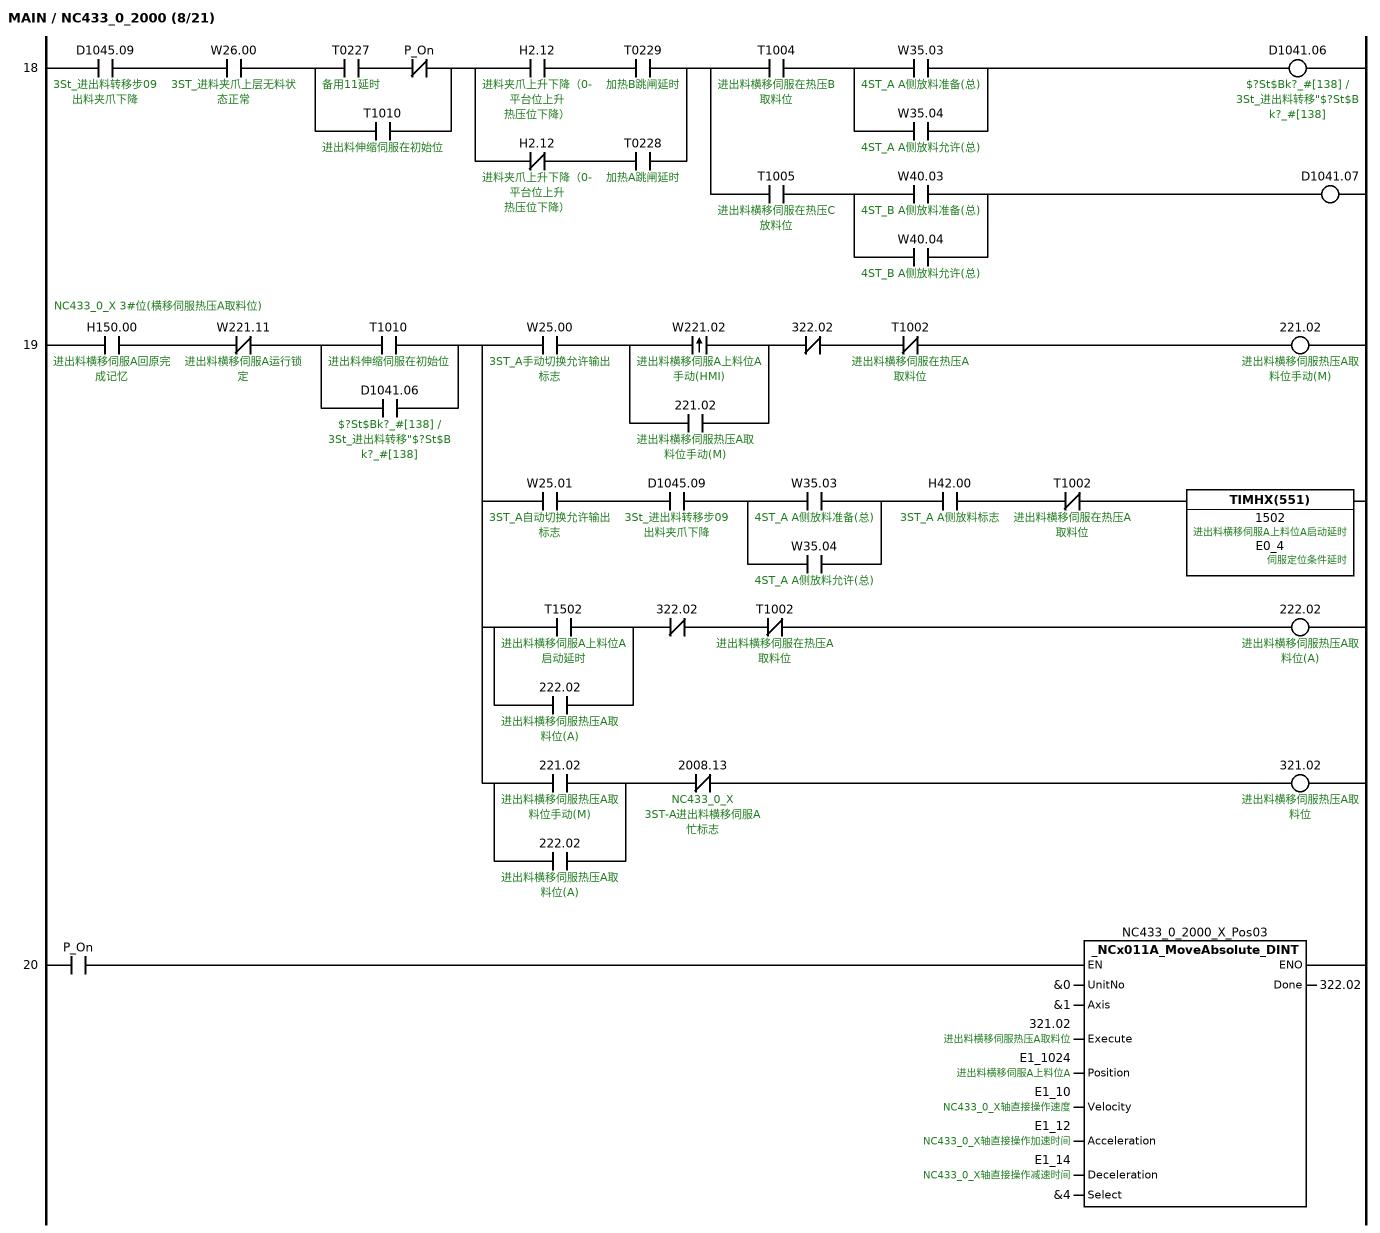
; rung 18
LD D1045.09  ; 3St_进出料转移步09 出料夹爪下降
AND W26.00  ; 3ST_进料夹爪上层无料状态正常
LD T0227  ; 备用11延时
ANDNOT P_On
OR T1010  ; 进出料伸缩伺服在初始位
ANDLD
LD H2.12  ; 进料夹爪上升下降（0-平台位上升  热压位下降）
AND T0229  ; 加热B跳闸延时
LDNOT H2.12  ; 进料夹爪上升下降（0-平台位上升  热压位下降）
AND T0228  ; 加热A跳闸延时
ORLD
ANDLD
OUT TR0
AND T1004  ; 进出料横移伺服在热压B取料位
LD W35.03  ; 4ST_A A侧放料准备(总)
OR W35.04  ; 4ST_A A侧放料允许(总)
ANDLD
OUT D1041.06  ; $?St$Bk?_#[138] / 3St_进出料转移"$?St$Bk?_#[138]
LD TR0
AND T1005  ; 进出料横移伺服在热压C放料位
LD W40.03  ; 4ST_B A侧放料准备(总)
OR W40.04  ; 4ST_B A侧放料允许(总)
ANDLD
OUT D1041.07
; rung 19: NC433_0_X 3#位(横移伺服热压A取料位)
LD H150.00  ; 进出料横移伺服A回原完成记忆
ANDNOT W221.11  ; 进出料横移伺服A运行锁定
LD T1010  ; 进出料伸缩伺服在初始位
OR D1041.06  ; $?St$Bk?_#[138] / 3St_进出料转移"$?St$Bk?_#[138]
ANDLD
OUT TR0
AND W25.00  ; 3ST_A手动切换允许输出标志
@LD W221.02  ; 进出料横移伺服A上料位A手动(HMI)
OR 221.02  ; 进出料横移伺服热压A取料位手动(M)
ANDLD
ANDNOT 322.02
ANDNOT T1002  ; 进出料横移伺服在热压A取料位
OUT 221.02  ; 进出料横移伺服热压A取料位手动(M)
LD TR0
AND W25.01  ; 3ST_A自动切换允许输出标志
AND D1045.09  ; 3St_进出料转移步09 出料夹爪下降
LD W35.03  ; 4ST_A A侧放料准备(总)
OR W35.04  ; 4ST_A A侧放料允许(总)
ANDLD
AND H42.00  ; 3ST_A A侧放料标志
ANDNOT T1002  ; 进出料横移伺服在热压A取料位
TIMHX(551) 1502 E0_4  ; 伺服定位条件延时, 进出料横移伺服A上料位A启动延时
LD TR0
LD T1502  ; 进出料横移伺服A上料位A启动延时
OR 222.02  ; 进出料横移伺服热压A取料位(A)
ANDLD
ANDNOT 322.02
ANDNOT T1002  ; 进出料横移伺服在热压A取料位
OUT 222.02  ; 进出料横移伺服热压A取料位(A)
LD TR0
LD 221.02  ; 进出料横移伺服热压A取料位手动(M)
OR 222.02  ; 进出料横移伺服热压A取料位(A)
ANDLD
ANDNOT 2008.13  ; NC433_0_X 3ST-A进出料横移伺服A忙标志
OUT 321.02  ; 进出料横移伺服热压A取料位
; rung 20
LD P_On
CALL NC433_0_2000_X_Pos03 : _NCx011A_MoveAbsolute_DINT (UnitNo := &0, Axis := &1, Execute := 321.02, Position := E1_1024, Velocity := E1_10, Acceleration := E1_12, Deceleration := E1_14, Select := &4, Done => 322.02)  ; 进出料横移伺服热压A取料位, 进出料横移伺服A上料位A, NC433_0_X轴直接操作速度, NC433_0_X轴直接操作加速时间, NC433_0_X轴直接操作减速时间

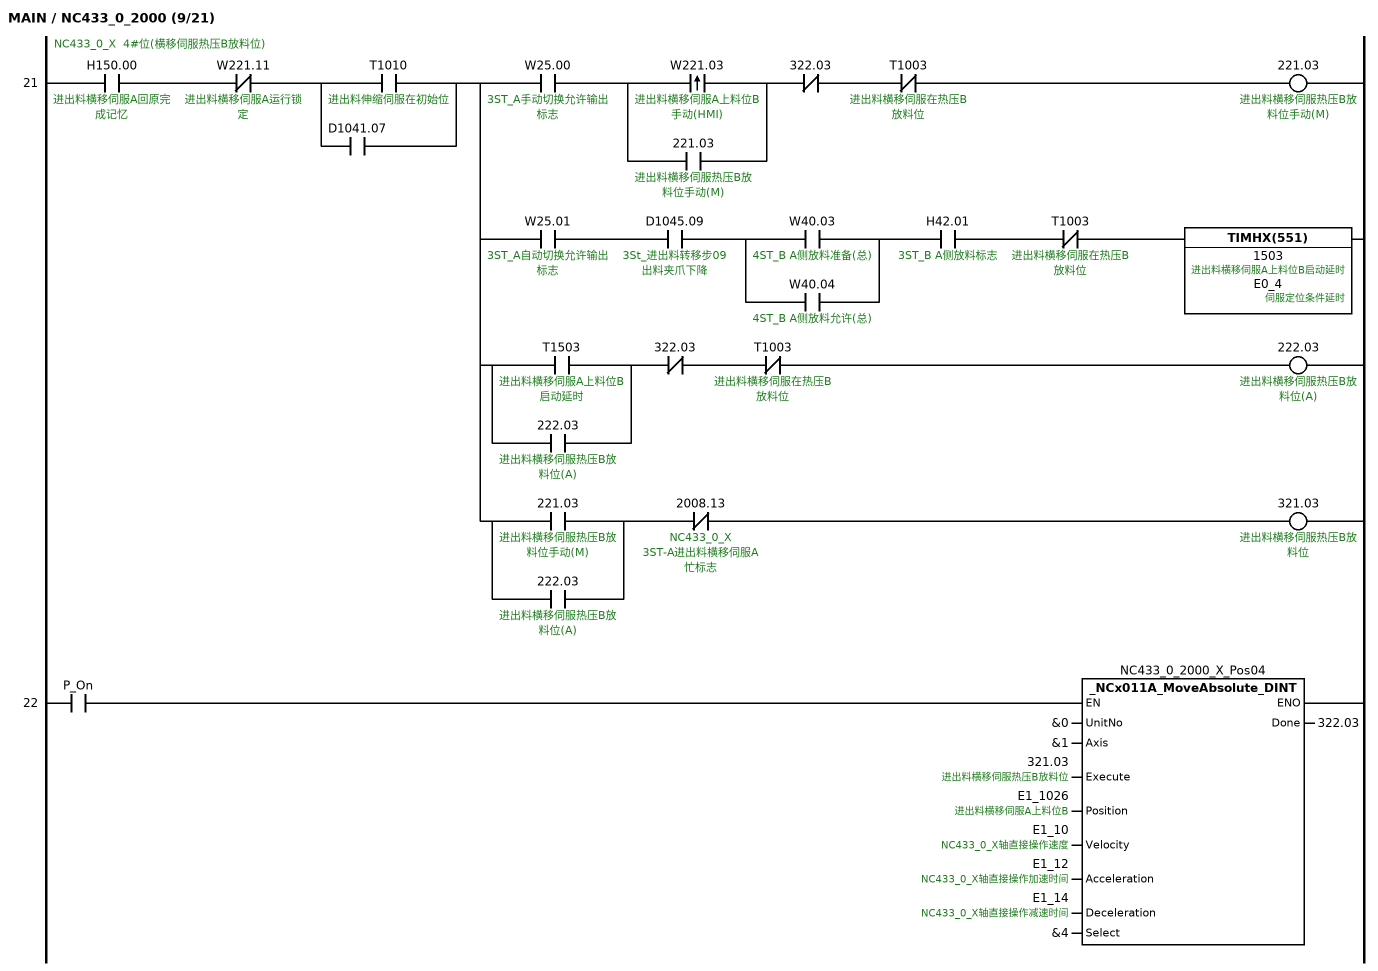
; rung 21: NC433_0_X  4#位(横移伺服热压B放料位)
LD H150.00  ; 进出料横移伺服A回原完成记忆
ANDNOT W221.11  ; 进出料横移伺服A运行锁定
LD T1010  ; 进出料伸缩伺服在初始位
OR D1041.07
ANDLD
OUT TR0
AND W25.00  ; 3ST_A手动切换允许输出标志
@LD W221.03  ; 进出料横移伺服A上料位B手动(HMI)
OR 221.03  ; 进出料横移伺服热压B放料位手动(M)
ANDLD
ANDNOT 322.03
ANDNOT T1003  ; 进出料横移伺服在热压B放料位
OUT 221.03  ; 进出料横移伺服热压B放料位手动(M)
LD TR0
AND W25.01  ; 3ST_A自动切换允许输出标志
AND D1045.09  ; 3St_进出料转移步09 出料夹爪下降
LD W40.03  ; 4ST_B A侧放料准备(总)
OR W40.04  ; 4ST_B A侧放料允许(总)
ANDLD
AND H42.01  ; 3ST_B A侧放料标志
ANDNOT T1003  ; 进出料横移伺服在热压B放料位
TIMHX(551) 1503 E0_4  ; 伺服定位条件延时, 进出料横移伺服A上料位B启动延时
LD TR0
LD T1503  ; 进出料横移伺服A上料位B启动延时
OR 222.03  ; 进出料横移伺服热压B放料位(A)
ANDLD
ANDNOT 322.03
ANDNOT T1003  ; 进出料横移伺服在热压B放料位
OUT 222.03  ; 进出料横移伺服热压B放料位(A)
LD TR0
LD 221.03  ; 进出料横移伺服热压B放料位手动(M)
OR 222.03  ; 进出料横移伺服热压B放料位(A)
ANDLD
ANDNOT 2008.13  ; NC433_0_X 3ST-A进出料横移伺服A忙标志
OUT 321.03  ; 进出料横移伺服热压B放料位
; rung 22
LD P_On
CALL NC433_0_2000_X_Pos04 : _NCx011A_MoveAbsolute_DINT (UnitNo := &0, Axis := &1, Execute := 321.03, Position := E1_1026, Velocity := E1_10, Acceleration := E1_12, Deceleration := E1_14, Select := &4, Done => 322.03)  ; 进出料横移伺服热压B放料位, 进出料横移伺服A上料位B, NC433_0_X轴直接操作速度, NC433_0_X轴直接操作加速时间, NC433_0_X轴直接操作减速时间

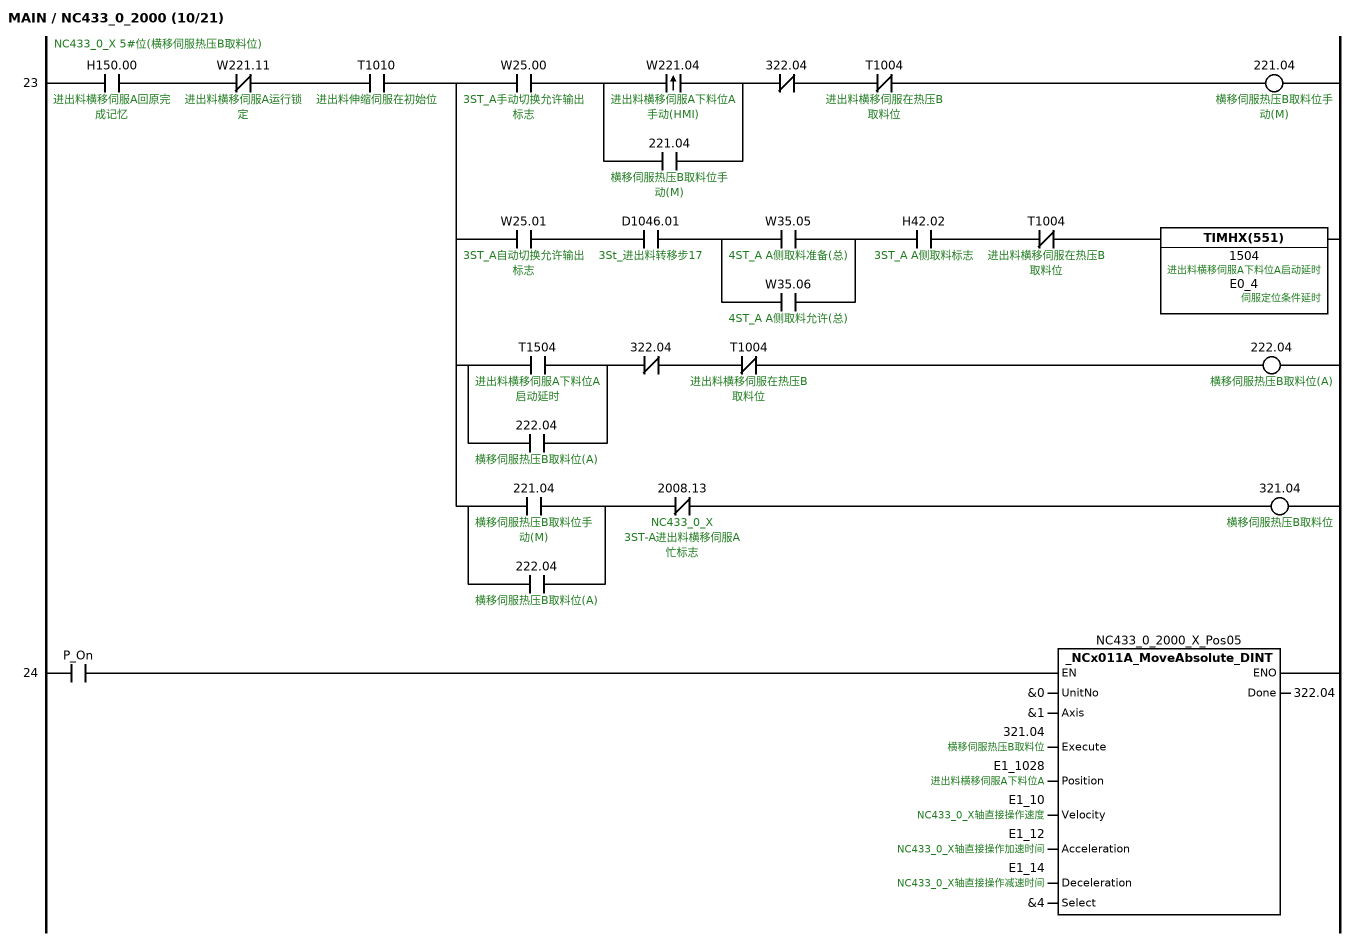
; rung 23: NC433_0_X 5#位(横移伺服热压B取料位)
LD H150.00  ; 进出料横移伺服A回原完成记忆
ANDNOT W221.11  ; 进出料横移伺服A运行锁定
AND T1010  ; 进出料伸缩伺服在初始位
OUT TR0
AND W25.00  ; 3ST_A手动切换允许输出标志
@LD W221.04  ; 进出料横移伺服A下料位A手动(HMI)
OR 221.04  ; 横移伺服热压B取料位手动(M)
ANDLD
ANDNOT 322.04
ANDNOT T1004  ; 进出料横移伺服在热压B取料位
OUT 221.04  ; 横移伺服热压B取料位手动(M)
LD TR0
AND W25.01  ; 3ST_A自动切换允许输出标志
AND D1046.01  ; 3St_进出料转移步17
LD W35.05  ; 4ST_A A侧取料准备(总)
OR W35.06  ; 4ST_A A侧取料允许(总)
ANDLD
AND H42.02  ; 3ST_A A侧取料标志
ANDNOT T1004  ; 进出料横移伺服在热压B取料位
TIMHX(551) 1504 E0_4  ; 伺服定位条件延时, 进出料横移伺服A下料位A启动延时
LD TR0
LD T1504  ; 进出料横移伺服A下料位A启动延时
OR 222.04  ; 横移伺服热压B取料位(A)
ANDLD
ANDNOT 322.04
ANDNOT T1004  ; 进出料横移伺服在热压B取料位
OUT 222.04  ; 横移伺服热压B取料位(A)
LD TR0
LD 221.04  ; 横移伺服热压B取料位手动(M)
OR 222.04  ; 横移伺服热压B取料位(A)
ANDLD
ANDNOT 2008.13  ; NC433_0_X 3ST-A进出料横移伺服A忙标志
OUT 321.04  ; 横移伺服热压B取料位
; rung 24
LD P_On
CALL NC433_0_2000_X_Pos05 : _NCx011A_MoveAbsolute_DINT (UnitNo := &0, Axis := &1, Execute := 321.04, Position := E1_1028, Velocity := E1_10, Acceleration := E1_12, Deceleration := E1_14, Select := &4, Done => 322.04)  ; 横移伺服热压B取料位, 进出料横移伺服A下料位A, NC433_0_X轴直接操作速度, NC433_0_X轴直接操作加速时间, NC433_0_X轴直接操作减速时间

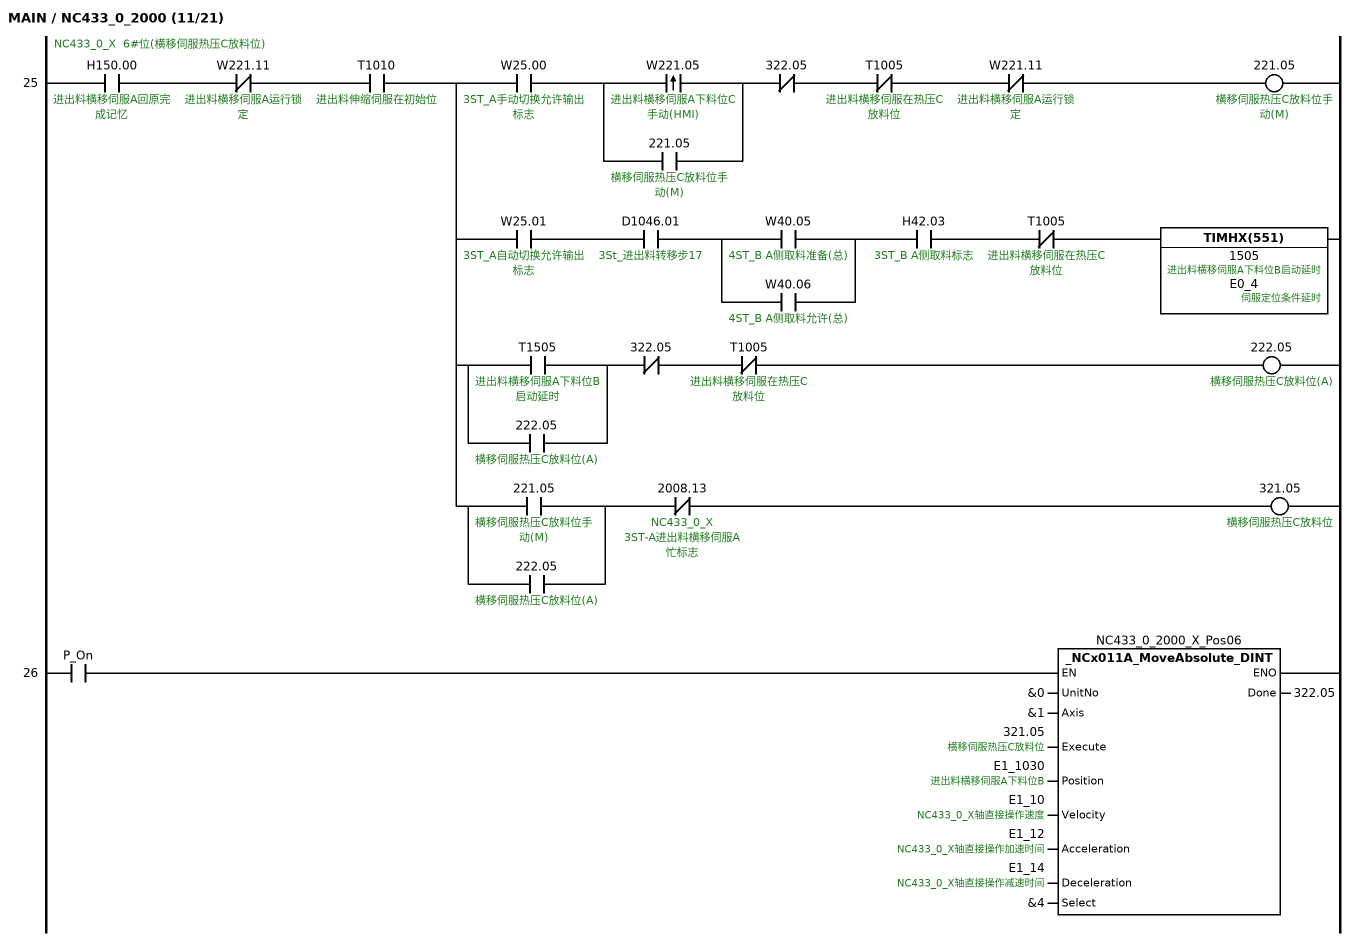
; rung 25: NC433_0_X  6#位(横移伺服热压C放料位)
LD H150.00  ; 进出料横移伺服A回原完成记忆
ANDNOT W221.11  ; 进出料横移伺服A运行锁定
AND T1010  ; 进出料伸缩伺服在初始位
OUT TR0
AND W25.00  ; 3ST_A手动切换允许输出标志
@LD W221.05  ; 进出料横移伺服A下料位C手动(HMI)
OR 221.05  ; 横移伺服热压C放料位手动(M)
ANDLD
ANDNOT 322.05
ANDNOT T1005  ; 进出料横移伺服在热压C放料位
ANDNOT W221.11  ; 进出料横移伺服A运行锁定
OUT 221.05  ; 横移伺服热压C放料位手动(M)
LD TR0
AND W25.01  ; 3ST_A自动切换允许输出标志
AND D1046.01  ; 3St_进出料转移步17
LD W40.05  ; 4ST_B A侧取料准备(总)
OR W40.06  ; 4ST_B A侧取料允许(总)
ANDLD
AND H42.03  ; 3ST_B A侧取料标志
ANDNOT T1005  ; 进出料横移伺服在热压C放料位
TIMHX(551) 1505 E0_4  ; 伺服定位条件延时, 进出料横移伺服A下料位B启动延时
LD TR0
LD T1505  ; 进出料横移伺服A下料位B启动延时
OR 222.05  ; 横移伺服热压C放料位(A)
ANDLD
ANDNOT 322.05
ANDNOT T1005  ; 进出料横移伺服在热压C放料位
OUT 222.05  ; 横移伺服热压C放料位(A)
LD TR0
LD 221.05  ; 横移伺服热压C放料位手动(M)
OR 222.05  ; 横移伺服热压C放料位(A)
ANDLD
ANDNOT 2008.13  ; NC433_0_X 3ST-A进出料横移伺服A忙标志
OUT 321.05  ; 横移伺服热压C放料位
; rung 26
LD P_On
CALL NC433_0_2000_X_Pos06 : _NCx011A_MoveAbsolute_DINT (UnitNo := &0, Axis := &1, Execute := 321.05, Position := E1_1030, Velocity := E1_10, Acceleration := E1_12, Deceleration := E1_14, Select := &4, Done => 322.05)  ; 横移伺服热压C放料位, 进出料横移伺服A下料位B, NC433_0_X轴直接操作速度, NC433_0_X轴直接操作加速时间, NC433_0_X轴直接操作减速时间

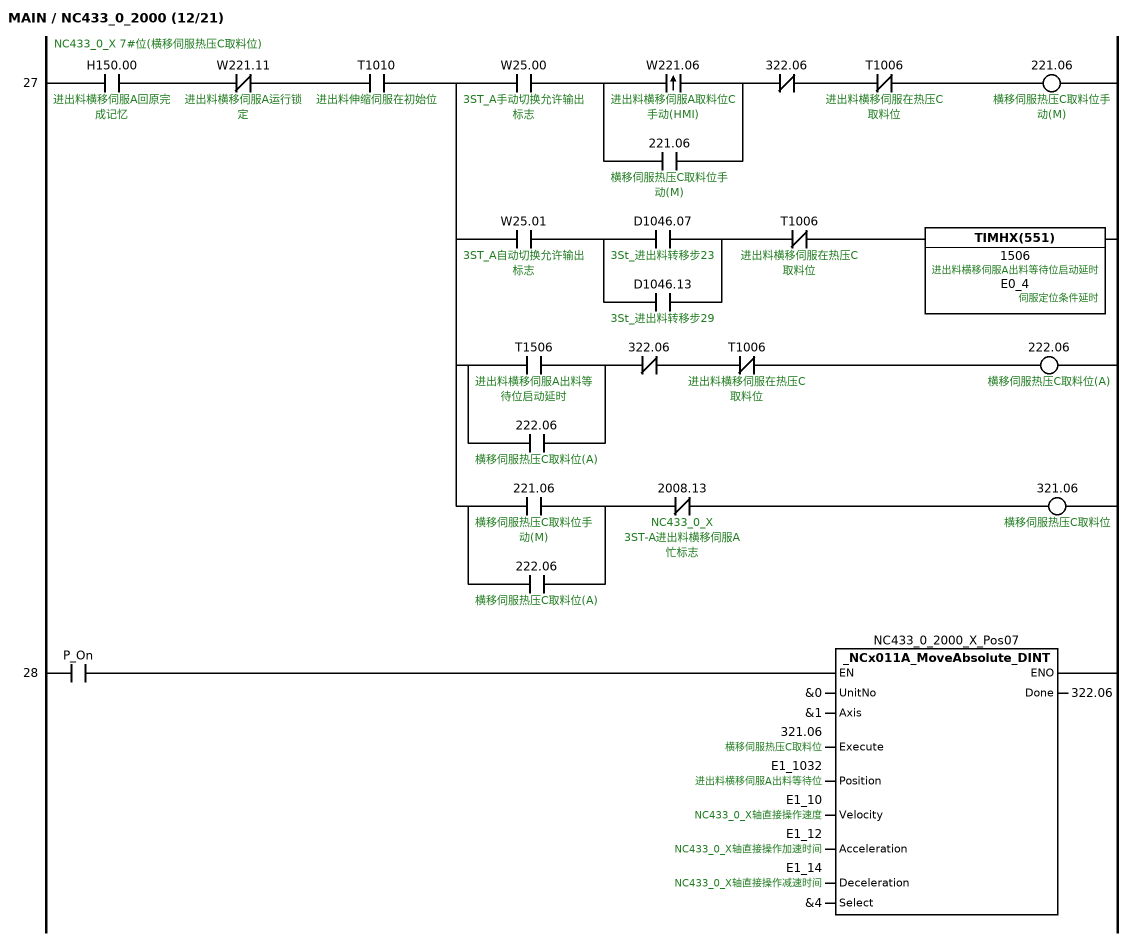
; rung 27: NC433_0_X 7#位(横移伺服热压C取料位)
LD H150.00  ; 进出料横移伺服A回原完成记忆
ANDNOT W221.11  ; 进出料横移伺服A运行锁定
AND T1010  ; 进出料伸缩伺服在初始位
OUT TR0
AND W25.00  ; 3ST_A手动切换允许输出标志
@LD W221.06  ; 进出料横移伺服A取料位C手动(HMI)
OR 221.06  ; 横移伺服热压C取料位手动(M)
ANDLD
ANDNOT 322.06
ANDNOT T1006  ; 进出料横移伺服在热压C取料位
OUT 221.06  ; 横移伺服热压C取料位手动(M)
LD TR0
AND W25.01  ; 3ST_A自动切换允许输出标志
LD D1046.07  ; 3St_进出料转移步23
OR D1046.13  ; 3St_进出料转移步29
ANDLD
ANDNOT T1006  ; 进出料横移伺服在热压C取料位
TIMHX(551) 1506 E0_4  ; 伺服定位条件延时, 进出料横移伺服A出料等待位启动延时
LD TR0
LD T1506  ; 进出料横移伺服A出料等待位启动延时
OR 222.06  ; 横移伺服热压C取料位(A)
ANDLD
ANDNOT 322.06
ANDNOT T1006  ; 进出料横移伺服在热压C取料位
OUT 222.06  ; 横移伺服热压C取料位(A)
LD TR0
LD 221.06  ; 横移伺服热压C取料位手动(M)
OR 222.06  ; 横移伺服热压C取料位(A)
ANDLD
ANDNOT 2008.13  ; NC433_0_X 3ST-A进出料横移伺服A忙标志
OUT 321.06  ; 横移伺服热压C取料位
; rung 28
LD P_On
CALL NC433_0_2000_X_Pos07 : _NCx011A_MoveAbsolute_DINT (UnitNo := &0, Axis := &1, Execute := 321.06, Position := E1_1032, Velocity := E1_10, Acceleration := E1_12, Deceleration := E1_14, Select := &4, Done => 322.06)  ; 横移伺服热压C取料位, 进出料横移伺服A出料等待位, NC433_0_X轴直接操作速度, NC433_0_X轴直接操作加速时间, NC433_0_X轴直接操作减速时间

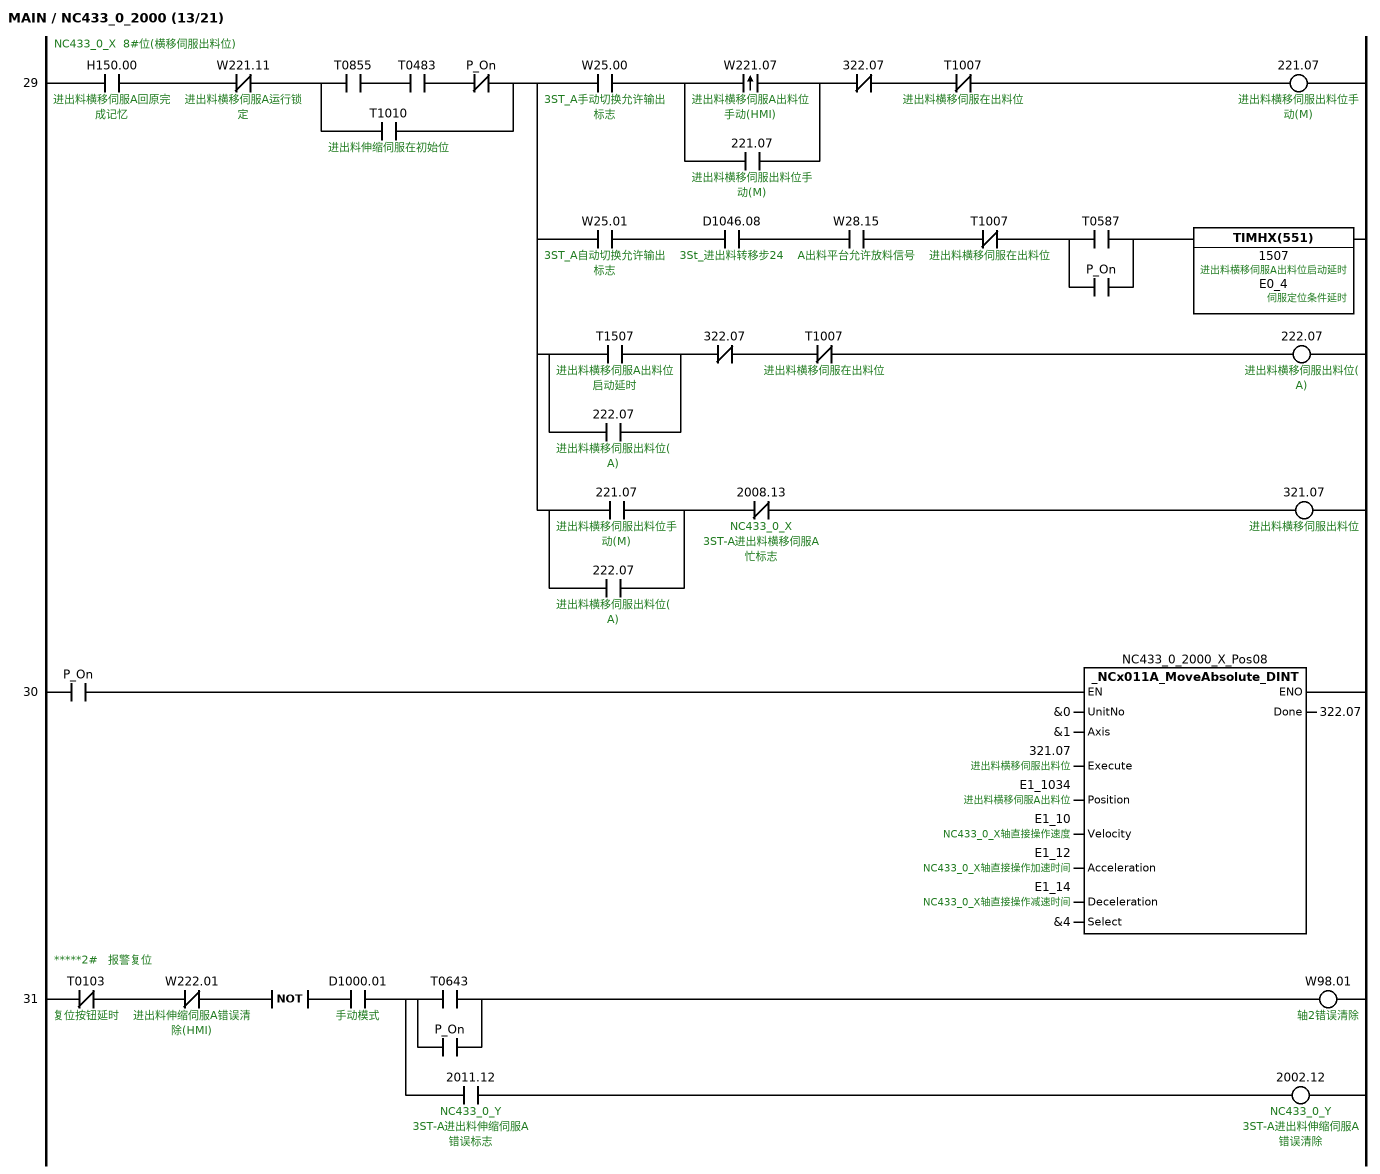
; rung 29: NC433_0_X  8#位(横移伺服出料位)
LD H150.00  ; 进出料横移伺服A回原完成记忆
ANDNOT W221.11  ; 进出料横移伺服A运行锁定
LD T0855
AND T0483
ANDNOT P_On
OR T1010  ; 进出料伸缩伺服在初始位
ANDLD
OUT TR0
AND W25.00  ; 3ST_A手动切换允许输出标志
@LD W221.07  ; 进出料横移伺服A出料位手动(HMI)
OR 221.07  ; 进出料横移伺服出料位手动(M)
ANDLD
ANDNOT 322.07
ANDNOT T1007  ; 进出料横移伺服在出料位
OUT 221.07  ; 进出料横移伺服出料位手动(M)
LD TR0
AND W25.01  ; 3ST_A自动切换允许输出标志
AND D1046.08  ; 3St_进出料转移步24
AND W28.15  ; A出料平台允许放料信号
ANDNOT T1007  ; 进出料横移伺服在出料位
LD T0587
OR P_On
ANDLD
TIMHX(551) 1507 E0_4  ; 伺服定位条件延时, 进出料横移伺服A出料位启动延时
LD TR0
LD T1507  ; 进出料横移伺服A出料位启动延时
OR 222.07  ; 进出料横移伺服出料位(A)
ANDLD
ANDNOT 322.07
ANDNOT T1007  ; 进出料横移伺服在出料位
OUT 222.07  ; 进出料横移伺服出料位(A)
LD TR0
LD 221.07  ; 进出料横移伺服出料位手动(M)
OR 222.07  ; 进出料横移伺服出料位(A)
ANDLD
ANDNOT 2008.13  ; NC433_0_X 3ST-A进出料横移伺服A忙标志
OUT 321.07  ; 进出料横移伺服出料位
; rung 30
LD P_On
CALL NC433_0_2000_X_Pos08 : _NCx011A_MoveAbsolute_DINT (UnitNo := &0, Axis := &1, Execute := 321.07, Position := E1_1034, Velocity := E1_10, Acceleration := E1_12, Deceleration := E1_14, Select := &4, Done => 322.07)  ; 进出料横移伺服出料位, 进出料横移伺服A出料位, NC433_0_X轴直接操作速度, NC433_0_X轴直接操作加速时间, NC433_0_X轴直接操作减速时间
; rung 31: *****2#   报警复位
LDNOT T0103  ; 复位按钮延时
ANDNOT W222.01  ; 进出料伸缩伺服A错误清除(HMI)
NOT(520)
AND D1000.01  ; 手动模式
OUT TR0
LD T0643
OR P_On
ANDLD
OUT W98.01  ; 轴2错误清除
LD TR0
AND 2011.12  ; NC433_0_Y 3ST-A进出料伸缩伺服A错误标志
OUT 2002.12  ; NC433_0_Y 3ST-A进出料伸缩伺服A错误清除

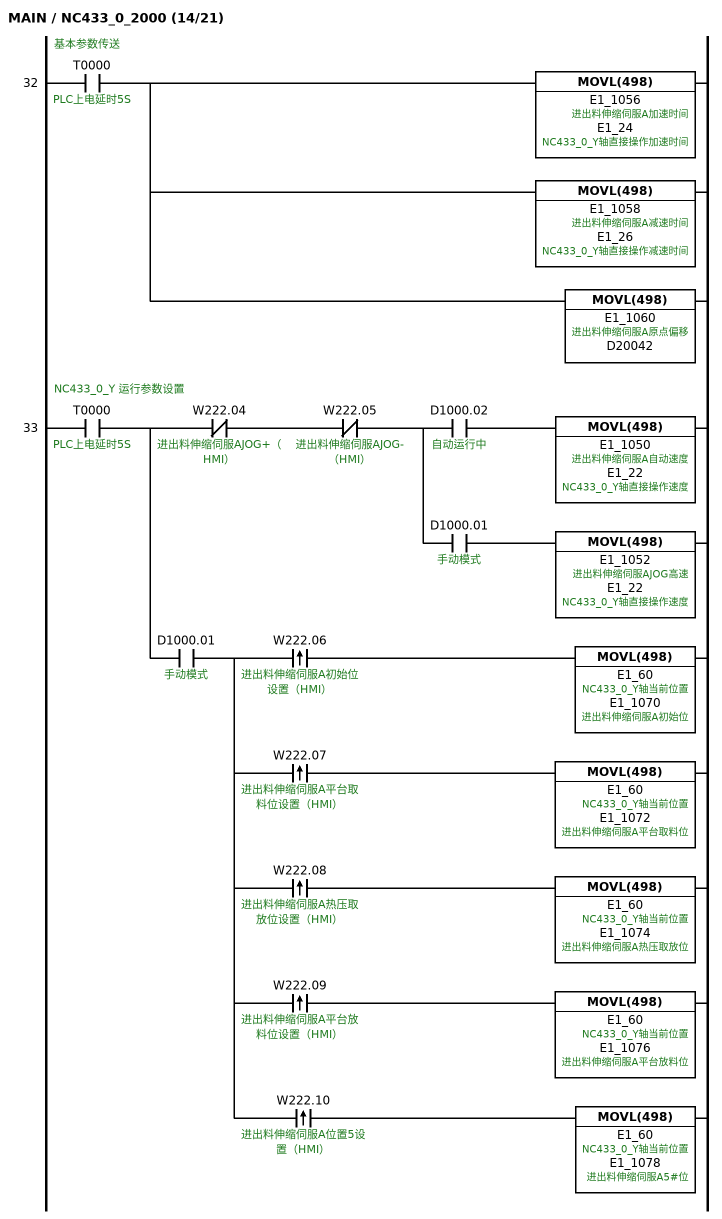
; rung 32: 基本参数传送
LD T0000  ; PLC上电延时5S
MOVL(498) E1_1056 E1_24  ; 进出料伸缩伺服A加速时间, NC433_0_Y轴直接操作加速时间
MOVL(498) E1_1058 E1_26  ; 进出料伸缩伺服A减速时间, NC433_0_Y轴直接操作减速时间
MOVL(498) E1_1060 D20042  ; 进出料伸缩伺服A原点偏移
; rung 33: NC433_0_Y 运行参数设置
LD T0000  ; PLC上电延时5S
OUT TR0
ANDNOT W222.04  ; 进出料伸缩伺服AJOG+（HMI）
ANDNOT W222.05  ; 进出料伸缩伺服AJOG-（HMI）
OUT TR1
AND D1000.02  ; 自动运行中
MOVL(498) E1_1050 E1_22  ; 进出料伸缩伺服A自动速度, NC433_0_Y轴直接操作速度
LD TR1
AND D1000.01  ; 手动模式
MOVL(498) E1_1052 E1_22  ; 进出料伸缩伺服AJOG高速, NC433_0_Y轴直接操作速度
LD TR0
AND D1000.01  ; 手动模式
OUT TR0
@AND W222.06  ; 进出料伸缩伺服A初始位设置（HMI）
MOVL(498) E1_60 E1_1070  ; NC433_0_Y轴当前位置, 进出料伸缩伺服A初始位
LD TR0
@AND W222.07  ; 进出料伸缩伺服A平台取料位设置（HMI）
MOVL(498) E1_60 E1_1072  ; NC433_0_Y轴当前位置, 进出料伸缩伺服A平台取料位
LD TR0
@AND W222.08  ; 进出料伸缩伺服A热压取放位设置（HMI）
MOVL(498) E1_60 E1_1074  ; NC433_0_Y轴当前位置, 进出料伸缩伺服A热压取放位
LD TR0
@AND W222.09  ; 进出料伸缩伺服A平台放料位设置（HMI）
MOVL(498) E1_60 E1_1076  ; NC433_0_Y轴当前位置, 进出料伸缩伺服A平台放料位
LD TR0
@AND W222.10  ; 进出料伸缩伺服A位置5设置（HMI）
MOVL(498) E1_60 E1_1078  ; NC433_0_Y轴当前位置, 进出料伸缩伺服A5#位

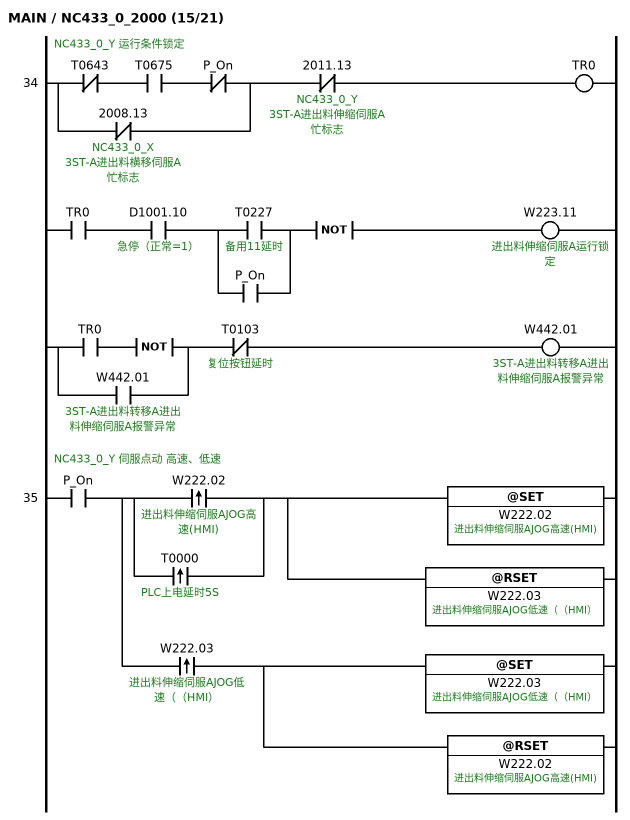
; rung 34: NC433_0_Y 运行条件锁定
LDNOT T0643
AND T0675
ANDNOT P_On
ORNOT 2008.13  ; NC433_0_X 3ST-A进出料横移伺服A忙标志
ANDNOT 2011.13  ; NC433_0_Y 3ST-A进出料伸缩伺服A忙标志
OUT TR0
AND D1001.10  ; 急停（正常=1）
LD T0227  ; 备用11延时
OR P_On
ANDLD
NOT(520)
OUT W223.11  ; 进出料伸缩伺服A运行锁定
LD TR0
NOT(520)
OR W442.01  ; 3ST-A进出料转移A进出料伸缩伺服A报警异常
ANDNOT T0103  ; 复位按钮延时
OUT W442.01  ; 3ST-A进出料转移A进出料伸缩伺服A报警异常
; rung 35: NC433_0_Y 伺服点动 高速、低速
LD P_On
OUT TR0
@LD W222.02  ; 进出料伸缩伺服AJOG高速(HMI)
@OR T0000  ; PLC上电延时5S
ANDLD
@SET W222.02  ; 进出料伸缩伺服AJOG高速(HMI)
@RSET W222.03  ; 进出料伸缩伺服AJOG低速（（HMI）
LD TR0
@AND W222.03  ; 进出料伸缩伺服AJOG低速（（HMI）
@SET W222.03  ; 进出料伸缩伺服AJOG低速（（HMI）
@RSET W222.02  ; 进出料伸缩伺服AJOG高速(HMI)

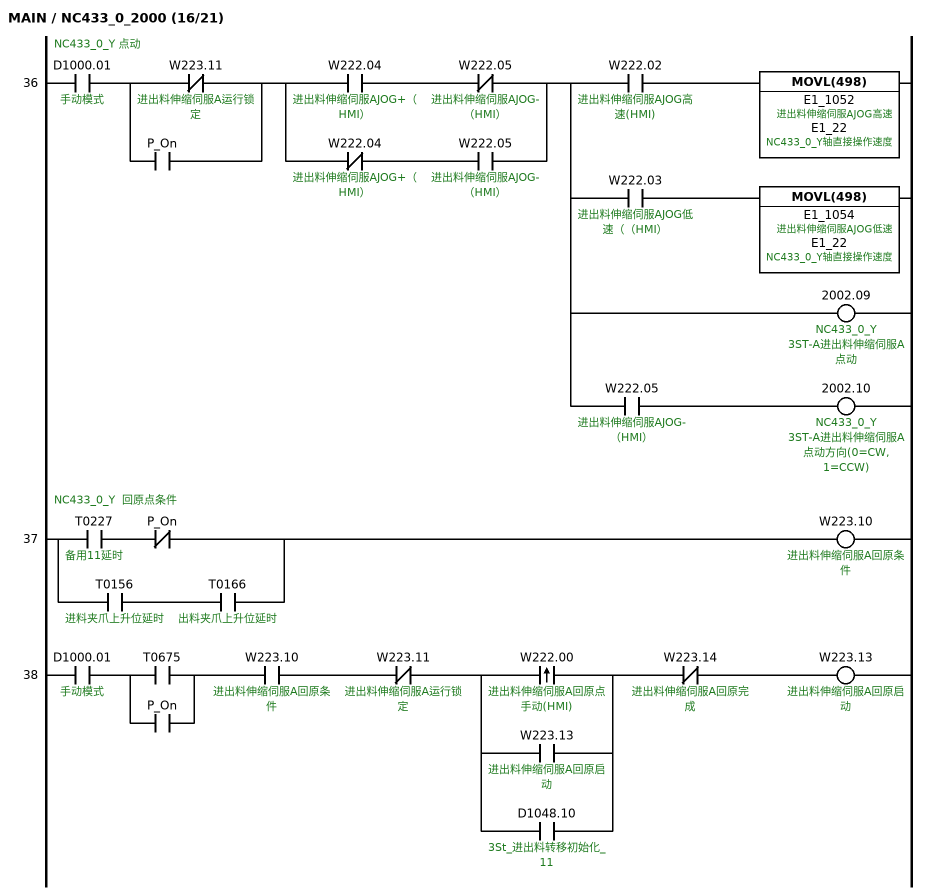
; rung 36: NC433_0_Y 点动
LD D1000.01  ; 手动模式
LDNOT W223.11  ; 进出料伸缩伺服A运行锁定
OR P_On
ANDLD
LD W222.04  ; 进出料伸缩伺服AJOG+（HMI）
ANDNOT W222.05  ; 进出料伸缩伺服AJOG-（HMI）
LDNOT W222.04  ; 进出料伸缩伺服AJOG+（HMI）
AND W222.05  ; 进出料伸缩伺服AJOG-（HMI）
ORLD
ANDLD
OUT TR0
AND W222.02  ; 进出料伸缩伺服AJOG高速(HMI)
MOVL(498) E1_1052 E1_22  ; 进出料伸缩伺服AJOG高速, NC433_0_Y轴直接操作速度
LD TR0
AND W222.03  ; 进出料伸缩伺服AJOG低速（（HMI）
MOVL(498) E1_1054 E1_22  ; 进出料伸缩伺服AJOG低速, NC433_0_Y轴直接操作速度
LD TR0
OUT 2002.09  ; NC433_0_Y 3ST-A进出料伸缩伺服A点动
AND W222.05  ; 进出料伸缩伺服AJOG-（HMI）
OUT 2002.10  ; NC433_0_Y 3ST-A进出料伸缩伺服A点动方向(0=CW,1=CCW)
; rung 37: NC433_0_Y  回原点条件
LD T0227  ; 备用11延时
ANDNOT P_On
LD T0156  ; 进料夹爪上升位延时
AND T0166  ; 出料夹爪上升位延时
ORLD
OUT W223.10  ; 进出料伸缩伺服A回原条件
; rung 38
LD D1000.01  ; 手动模式
LD T0675
OR P_On
ANDLD
AND W223.10  ; 进出料伸缩伺服A回原条件
ANDNOT W223.11  ; 进出料伸缩伺服A运行锁定
@LD W222.00  ; 进出料伸缩伺服A回原点手动(HMI)
OR W223.13  ; 进出料伸缩伺服A回原启动
OR D1048.10  ; 3St_进出料转移初始化_11
ANDLD
ANDNOT W223.14  ; 进出料伸缩伺服A回原完成
OUT W223.13  ; 进出料伸缩伺服A回原启动

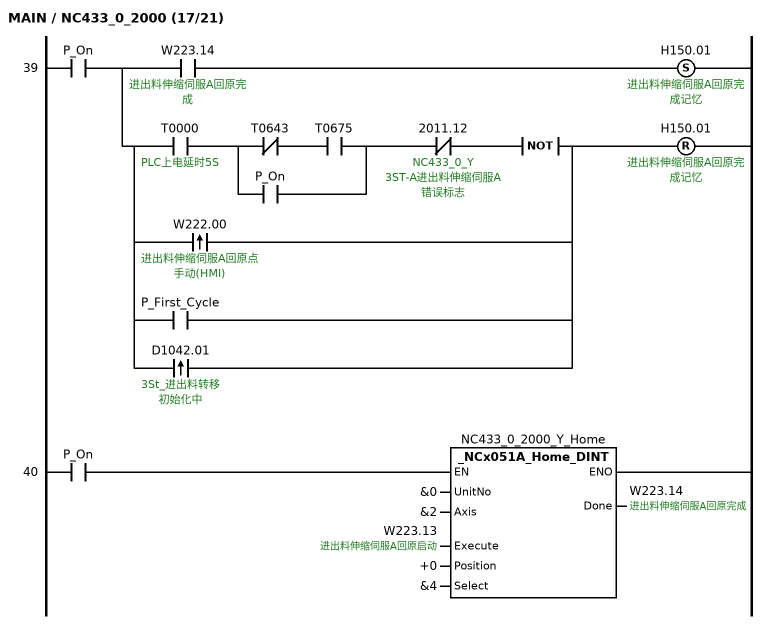
; rung 39
LD P_On
OUT TR0
AND W223.14  ; 进出料伸缩伺服A回原完成
SET H150.01  ; 进出料伸缩伺服A回原完成记忆
LD TR0
LD T0000  ; PLC上电延时5S
LDNOT T0643
AND T0675
OR P_On
ANDLD
ANDNOT 2011.12  ; NC433_0_Y 3ST-A进出料伸缩伺服A错误标志
NOT(520)
@OR W222.00  ; 进出料伸缩伺服A回原点手动(HMI)
OR P_First_Cycle
@OR D1042.01  ; 3St_进出料转移 初始化中
ANDLD
RSET H150.01  ; 进出料伸缩伺服A回原完成记忆
; rung 40
LD P_On
CALL NC433_0_2000_Y_Home : _NCx051A_Home_DINT (UnitNo := &0, Axis := &2, Execute := W223.13, Position := +0, Select := &4, Done => W223.14)  ; 进出料伸缩伺服A回原启动, 进出料伸缩伺服A回原完成

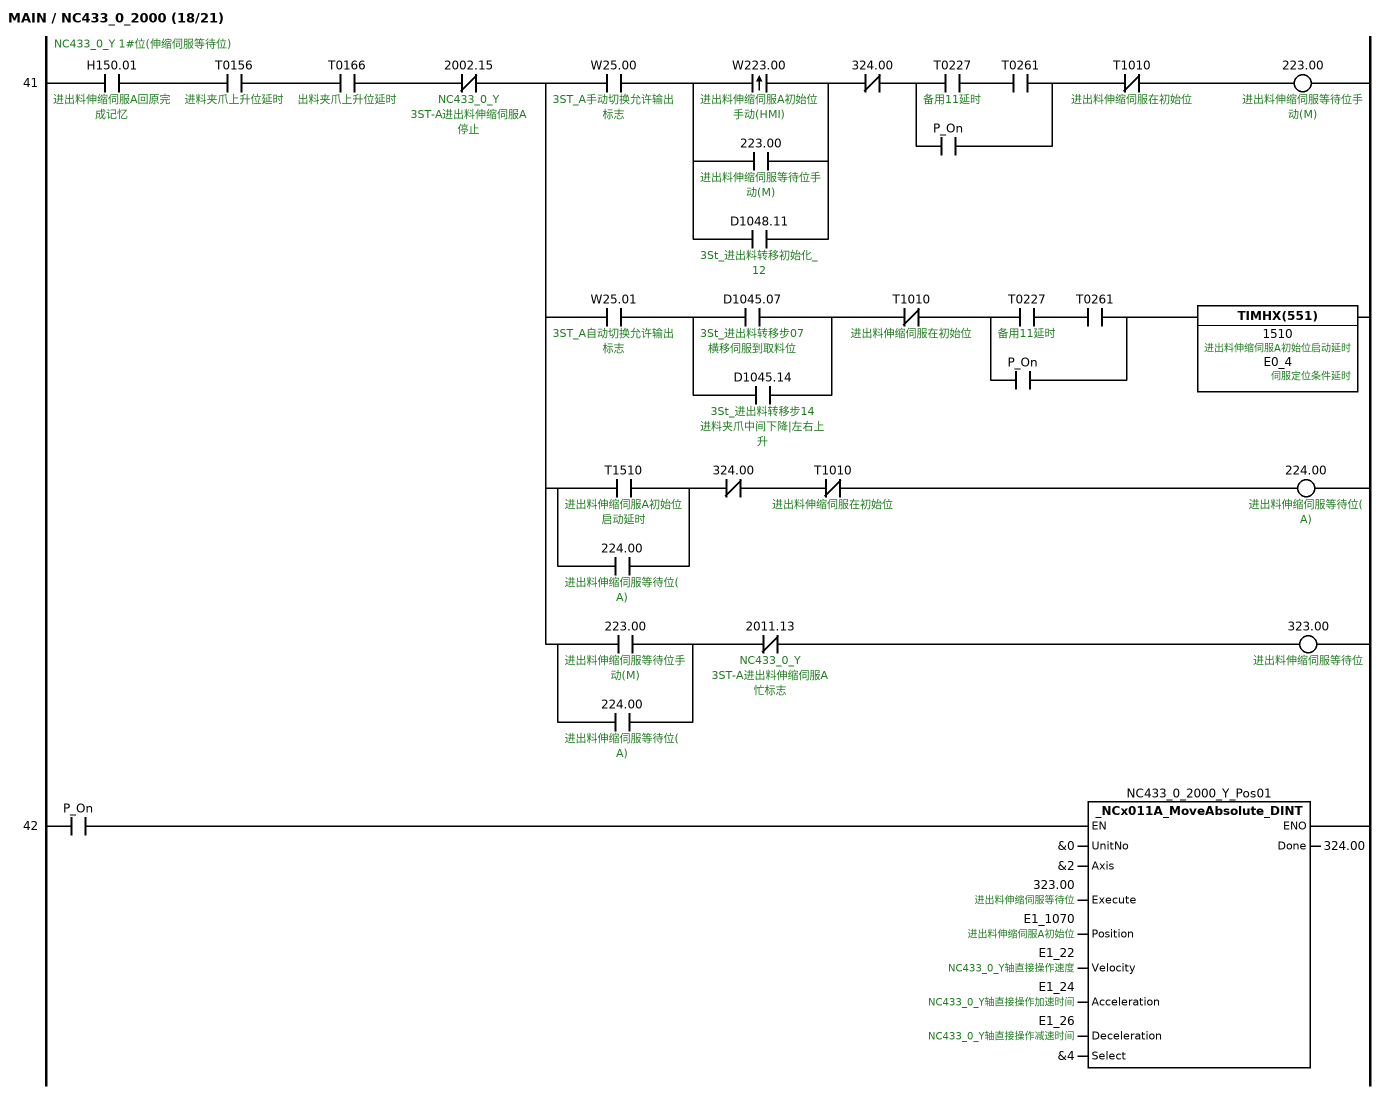
; rung 41: NC433_0_Y 1#位(伸缩伺服等待位)
LD H150.01  ; 进出料伸缩伺服A回原完成记忆
AND T0156  ; 进料夹爪上升位延时
AND T0166  ; 出料夹爪上升位延时
ANDNOT 2002.15  ; NC433_0_Y 3ST-A进出料伸缩伺服A停止
OUT TR0
AND W25.00  ; 3ST_A手动切换允许输出标志
@LD W223.00  ; 进出料伸缩伺服A初始位手动(HMI)
OR 223.00  ; 进出料伸缩伺服等待位手动(M)
OR D1048.11  ; 3St_进出料转移初始化_12
ANDLD
ANDNOT 324.00
LD T0227  ; 备用11延时
AND T0261
OR P_On
ANDLD
ANDNOT T1010  ; 进出料伸缩伺服在初始位
OUT 223.00  ; 进出料伸缩伺服等待位手动(M)
LD TR0
AND W25.01  ; 3ST_A自动切换允许输出标志
LD D1045.07  ; 3St_进出料转移步07 横移伺服到取料位
OR D1045.14  ; 3St_进出料转移步14 进料夹爪中间下降|左右上升
ANDLD
ANDNOT T1010  ; 进出料伸缩伺服在初始位
LD T0227  ; 备用11延时
AND T0261
OR P_On
ANDLD
TIMHX(551) 1510 E0_4  ; 伺服定位条件延时, 进出料伸缩伺服A初始位启动延时
LD TR0
LD T1510  ; 进出料伸缩伺服A初始位启动延时
OR 224.00  ; 进出料伸缩伺服等待位(A)
ANDLD
ANDNOT 324.00
ANDNOT T1010  ; 进出料伸缩伺服在初始位
OUT 224.00  ; 进出料伸缩伺服等待位(A)
LD TR0
LD 223.00  ; 进出料伸缩伺服等待位手动(M)
OR 224.00  ; 进出料伸缩伺服等待位(A)
ANDLD
ANDNOT 2011.13  ; NC433_0_Y 3ST-A进出料伸缩伺服A忙标志
OUT 323.00  ; 进出料伸缩伺服等待位
; rung 42
LD P_On
CALL NC433_0_2000_Y_Pos01 : _NCx011A_MoveAbsolute_DINT (UnitNo := &0, Axis := &2, Execute := 323.00, Position := E1_1070, Velocity := E1_22, Acceleration := E1_24, Deceleration := E1_26, Select := &4, Done => 324.00)  ; 进出料伸缩伺服等待位, 进出料伸缩伺服A初始位, NC433_0_Y轴直接操作速度, NC433_0_Y轴直接操作加速时间, NC433_0_Y轴直接操作减速时间

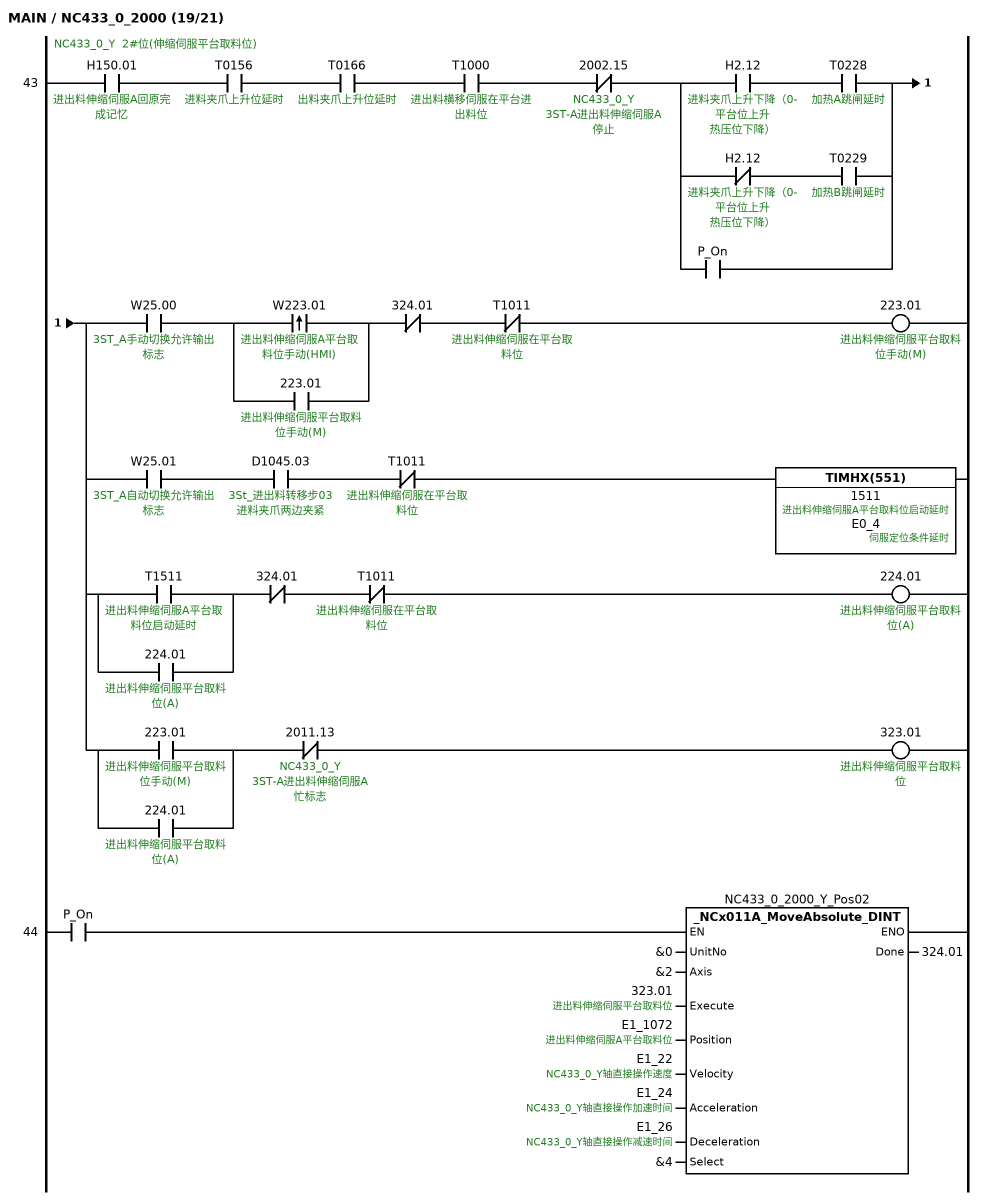
; rung 43: NC433_0_Y  2#位(伸缩伺服平台取料位)
LD H150.01  ; 进出料伸缩伺服A回原完成记忆
AND T0156  ; 进料夹爪上升位延时
AND T0166  ; 出料夹爪上升位延时
AND T1000  ; 进出料横移伺服在平台进出料位
ANDNOT 2002.15  ; NC433_0_Y 3ST-A进出料伸缩伺服A停止
LD H2.12  ; 进料夹爪上升下降（0-平台位上升  热压位下降）
AND T0228  ; 加热A跳闸延时
LDNOT H2.12  ; 进料夹爪上升下降（0-平台位上升  热压位下降）
AND T0229  ; 加热B跳闸延时
ORLD
OR P_On
ANDLD
OUT TR0
AND W25.00  ; 3ST_A手动切换允许输出标志
@LD W223.01  ; 进出料伸缩伺服A平台取料位手动(HMI)
OR 223.01  ; 进出料伸缩伺服平台取料位手动(M)
ANDLD
ANDNOT 324.01
ANDNOT T1011  ; 进出料伸缩伺服在平台取料位
OUT 223.01  ; 进出料伸缩伺服平台取料位手动(M)
LD TR0
AND W25.01  ; 3ST_A自动切换允许输出标志
AND D1045.03  ; 3St_进出料转移步03 进料夹爪两边夹紧
ANDNOT T1011  ; 进出料伸缩伺服在平台取料位
TIMHX(551) 1511 E0_4  ; 伺服定位条件延时, 进出料伸缩伺服A平台取料位启动延时
LD TR0
LD T1511  ; 进出料伸缩伺服A平台取料位启动延时
OR 224.01  ; 进出料伸缩伺服平台取料位(A)
ANDLD
ANDNOT 324.01
ANDNOT T1011  ; 进出料伸缩伺服在平台取料位
OUT 224.01  ; 进出料伸缩伺服平台取料位(A)
LD TR0
LD 223.01  ; 进出料伸缩伺服平台取料位手动(M)
OR 224.01  ; 进出料伸缩伺服平台取料位(A)
ANDLD
ANDNOT 2011.13  ; NC433_0_Y 3ST-A进出料伸缩伺服A忙标志
OUT 323.01  ; 进出料伸缩伺服平台取料位
; rung 44
LD P_On
CALL NC433_0_2000_Y_Pos02 : _NCx011A_MoveAbsolute_DINT (UnitNo := &0, Axis := &2, Execute := 323.01, Position := E1_1072, Velocity := E1_22, Acceleration := E1_24, Deceleration := E1_26, Select := &4, Done => 324.01)  ; 进出料伸缩伺服平台取料位, 进出料伸缩伺服A平台取料位, NC433_0_Y轴直接操作速度, NC433_0_Y轴直接操作加速时间, NC433_0_Y轴直接操作减速时间

